C09126=1020.009,-60.580,383.207,-24.059,21.610,-43.700
C09127=1020.010,-60.243,383.182,-24.060,21.610,-43.695
C09128=1020.011,-59.906,383.156,-24.060,21.609,-43.691
C09129=1020.011,-59.569,383.131,-24.061,21.609,-43.686
C09130=1020.011,-59.234,383.106,-24.062,21.608,-43.680
C09131=1020.012,-58.898,383.081,-24.062,21.608,-43.676
C09132=1020.012,-58.562,383.056,-24.063,21.607,-43.671
C09133=1020.013,-58.228,383.030,-24.064,21.607,-43.666
C09134=1020.014,-57.893,383.005,-24.064,21.606,-43.662
C09135=1020.014,-57.559,382.981,-24.065,21.606,-43.656
C09136=1020.014,-57.225,382.955,-24.066,21.605,-43.652
C09137=1020.015,-56.892,382.930,-24.066,21.604,-43.647
C09138=1020.015,-56.558,382.905,-24.067,21.605,-43.642
C09139=1020.017,-56.225,382.880,-24.068,21.603,-43.637
C09140=1020.017,-55.892,382.855,-24.068,21.603,-43.632
C09141=1020.017,-55.559,382.830,-24.069,21.603,-43.627
C09142=1020.018,-55.226,382.805,-24.070,21.602,-43.623
C09143=1020.018,-54.894,382.780,-24.070,21.602,-43.618
C09144=1020.019,-54.562,382.755,-24.071,21.601,-43.613
C09145=1020.019,-54.229,382.729,-24.072,21.601,-43.608
C09146=1020.019,-53.896,382.704,-24.072,21.600,-43.603
C09147=1020.020,-53.565,382.679,-24.073,21.599,-43.599
C09148=1020.020,-53.232,382.654,-24.074,21.600,-43.594
C09149=1020.021,-52.900,382.629,-24.074,21.598,-43.589
C09150=1020.021,-52.568,382.604,-24.075,21.598,-43.584
C09151=1020.021,-52.235,382.579,-24.075,21.597,-43.579
C09152=1020.022,-51.903,382.554,-24.076,21.597,-43.575
C09153=1020.022,-51.571,382.528,-24.077,21.597,-43.570
C09154=1020.022,-51.238,382.503,-24.077,21.596,-43.566
C09155=1020.023,-50.906,382.478,-24.078,21.596,-43.560
C09156=1020.023,-50.524,382.449,-24.079,21.595,-43.555
C09157=1020.012,-29.274,380.804,-24.119,21.564,-43.254
C09158=1020.012,-28.955,380.779,-24.119,21.563,-43.250
C09159=1020.011,-28.621,380.753,-24.120,21.563,-43.245
C09160=1020.011,-28.288,380.727,-24.120,21.562,-43.241
C09161=1020.010,-27.956,380.700,-24.121,21.562,-43.236
C09162=1020.009,-27.623,380.673,-24.122,21.562,-43.232
C09163=1020.009,-27.291,380.647,-24.123,21.562,-43.227
C09164=1020.008,-26.957,380.622,-24.123,21.560,-43.223
C09165=1020.007,-26.625,380.595,-24.124,21.560,-43.217
C09166=1020.007,-26.292,380.569,-24.124,21.560,-43.214
C09167=1020.006,-25.960,380.542,-24.125,21.559,-43.208
C09168=1020.005,-25.627,380.516,-24.126,21.559,-43.204
C09169=1020.004,-25.294,380.490,-24.126,21.559,-43.199
C09170=1020.004,-24.960,380.463,-24.127,21.558,-43.195
C09171=1020.003,-24.628,380.437,-24.128,21.558,-43.190
C09172=1020.003,-24.295,380.410,-24.128,21.557,-43.186
C09173=1020.001,-23.963,380.384,-24.129,21.557,-43.181
C09174=1020.001,-23.630,380.357,-24.129,21.556,-43.177
C09175=1020.000,-23.297,380.332,-24.130,21.556,-43.171
C09176=1019.999,-22.964,380.305,-24.131,21.555,-43.168
C09177=1019.998,-22.632,380.279,-24.131,21.556,-43.162
C09178=1019.997,-22.299,380.252,-24.132,21.554,-43.158
C09179=1019.996,-21.966,380.225,-24.133,21.554,-43.153
C09180=1019.995,-21.633,380.198,-24.133,21.554,-43.149
C09181=1019.995,-21.301,380.172,-24.134,21.553,-43.144
C09182=1019.993,-20.967,380.146,-24.134,21.552,-43.140
C09183=1019.993,-20.634,380.119,-24.135,21.553,-43.135
C09184=1019.992,-20.301,380.093,-24.136,21.552,-43.131
C09185=1019.991,-19.969,380.066,-24.136,21.551,-43.127
C09186=1019.990,-19.636,380.039,-24.137,21.551,-43.122
C09187=1019.990,-19.464,380.025,-24.137,21.550,-43.118
C09188=1019.989,-19.048,379.992,-24.138,21.550,-43.112
C09189=1019.987,-18.800,379.973,-24.139,21.550,-43.109
C09190=1019.987,-18.538,379.952,-24.139,21.550,-43.107
C09191=1019.986,-18.276,379.931,-24.139,21.549,-43.105
C09192=1019.985,-18.029,379.911,-24.139,21.548,-43.103
C09193=1019.984,-17.807,379.893,-24.140,21.549,-43.100
C09194=1019.984,-17.442,379.864,-24.141,21.548,-43.092
C09195=1019.982,-17.109,379.837,-24.141,21.547,-43.088
C09196=1019.981,-16.776,379.811,-24.142,21.547,-43.083
C09197=1019.980,-16.442,379.783,-24.142,21.547,-43.079
C09198=1019.979,-16.109,379.757,-24.143,21.546,-43.074
C09199=1019.978,-15.775,379.730,-24.144,21.546,-43.070
C09200=1019.977,-15.439,379.703,-24.145,21.546,-43.065
C09201=1019.976,-15.103,379.676,-24.145,21.545,-43.061
C09202=1019.975,-14.765,379.649,-24.146,21.544,-43.055
C09203=1019.974,-14.425,379.622,-24.146,21.544,-43.052
C09204=1019.972,-14.083,379.593,-24.147,21.544,-43.046
C09205=1019.970,-13.739,379.566,-24.147,21.543,-43.042
C09206=1019.970,-13.392,379.538,-24.148,21.543,-43.037
C09207=1019.969,-13.044,379.510,-24.149,21.542,-43.033
C09208=1019.967,-12.694,379.481,-24.149,21.542,-43.028
C09209=1019.966,-12.342,379.453,-24.150,21.541,-43.024
C09210=1019.965,-11.989,379.425,-24.151,21.541,-43.019
C09211=1019.964,-11.633,379.396,-24.151,21.540,-43.014
C09212=1019.962,-11.277,379.367,-24.152,21.540,-43.009
C09213=1019.961,-10.919,379.338,-24.152,21.539,-43.006
C09214=1019.959,-10.560,379.309,-24.153,21.539,-43.000
C09215=1019.958,-10.200,379.280,-24.154,21.539,-42.995
C09216=1019.957,-9.839,379.251,-24.154,21.538,-42.991
C09217=1019.955,-9.478,379.222,-24.155,21.538,-42.985
C09218=1019.953,-9.115,379.192,-24.156,21.537,-42.982
C09219=1019.951,-8.753,379.163,-24.156,21.536,-42.976
C09220=1019.951,-8.390,379.134,-24.157,21.536,-42.971
C09221=1019.949,-8.027,379.104,-24.158,21.536,-42.967
C09222=1019.947,-7.664,379.074,-24.158,21.535,-42.961
C09223=1019.946,-7.298,379.045,-24.159,21.535,-42.956
C09224=1019.944,-6.929,379.014,-24.160,21.534,-42.952
C09225=1019.942,-6.557,378.984,-24.160,21.534,-42.947
C09226=1019.941,-6.183,378.954,-24.161,21.533,-42.941
C09227=1019.939,-5.806,378.923,-24.162,21.533,-42.937
C09228=1019.937,-5.431,378.893,-24.163,21.533,-42.932
C09229=1019.936,-5.058,378.862,-24.163,21.532,-42.928
C09230=1019.934,-4.687,378.831,-24.164,21.532,-42.923
C09231=1019.932,-4.322,378.802,-24.164,21.531,-42.919
C09232=1019.931,-3.961,378.772,-24.165,21.530,-42.913
C09233=1019.929,-3.602,378.743,-24.166,21.531,-42.908
C09234=1019.927,-3.249,378.714,-24.166,21.529,-42.904
C09235=1019.926,-2.896,378.685,-24.167,21.529,-42.899
C09236=1019.924,-2.544,378.656,-24.167,21.529,-42.895
C09237=1019.922,-2.195,378.627,-24.168,21.529,-42.890
C09238=1019.920,-1.846,378.599,-24.169,21.528,-42.886
C09239=1019.918,-1.500,378.571,-24.169,21.528,-42.880
C09240=1019.917,-1.155,378.542,-24.170,21.527,-42.877
C09241=1019.916,-0.811,378.514,-24.170,21.527,-42.873
C09242=1019.914,-0.469,378.486,-24.171,21.526,-42.867
C09243=1019.912,-0.129,378.458,-24.172,21.526,-42.864
C09244=1019.910,0.209,378.430,-24.172,21.526,-42.858
C09245=1019.909,0.546,378.403,-24.173,21.525,-42.855
C09246=1019.907,0.882,378.375,-24.173,21.525,-42.851
C09247=1019.906,1.217,378.348,-24.174,21.525,-42.846
C09248=1019.903,1.551,378.320,-24.175,21.524,-42.842
C09249=1019.901,1.885,378.293,-24.175,21.523,-42.838
C09250=1019.900,2.215,378.266,-24.176,21.523,-42.834
C09251=1019.898,2.528,378.239,-24.176,21.523,-42.831
C09252=1019.897,2.816,378.215,-24.177,21.522,-42.827
C09253=1019.895,3.085,378.194,-24.177,21.522,-42.823
C09254=1019.894,3.347,378.172,-24.178,21.522,-42.818
C09255=1019.892,3.616,378.150,-24.179,21.521,-42.814
C09256=1019.890,3.905,378.126,-24.179,21.521,-42.810
C09257=1019.889,4.218,378.100,-24.179,21.520,-42.807
C09258=1019.887,4.548,378.073,-24.180,21.521,-42.803
C09259=1019.884,4.880,378.045,-24.180,21.519,-42.799
C09260=1019.883,5.211,378.018,-24.181,21.519,-42.795
C09261=1019.881,5.541,377.990,-24.181,21.518,-42.792
C09262=1019.879,5.872,377.963,-24.182,21.519,-42.786
C09263=1019.877,6.202,377.936,-24.183,21.518,-42.783
C09264=1019.876,6.531,377.909,-24.183,21.518,-42.779
C09265=1019.873,6.860,377.881,-24.184,21.518,-42.774
C09266=1019.872,7.189,377.854,-24.185,21.517,-42.770
C09267=1019.870,7.516,377.827,-24.185,21.517,-42.766
C09268=1019.867,7.842,377.799,-24.186,21.516,-42.762
C09269=1019.866,8.165,377.773,-24.186,21.516,-42.759
C09270=1019.864,8.486,377.746,-24.186,21.515,-42.755
C09271=1019.862,8.804,377.720,-24.187,21.516,-42.750
C09272=1019.860,9.120,377.694,-24.188,21.515,-42.746
C09273=1019.858,9.436,377.668,-24.188,21.515,-42.742
C09274=1019.856,9.750,377.641,-24.189,21.514,-42.738
C09275=1019.854,10.065,377.615,-24.190,21.514,-42.733
C09276=1019.852,10.380,377.589,-24.190,21.514,-42.730
C09277=1019.850,10.698,377.562,-24.191,21.513,-42.726
C09278=1019.848,11.016,377.535,-24.191,21.513,-42.722
C09279=1019.846,11.337,377.509,-24.192,21.512,-42.718
C09280=1019.843,11.659,377.482,-24.192,21.512,-42.715
C09281=1019.842,11.982,377.455,-24.193,21.511,-42.711
C09282=1019.840,12.306,377.428,-24.193,21.511,-42.707
C09283=1019.837,12.630,377.401,-24.194,21.511,-42.702
C09284=1019.835,12.953,377.374,-24.194,21.510,-42.698
C09285=1019.833,13.277,377.346,-24.195,21.510,-42.694
C09286=1019.831,13.601,377.320,-24.195,21.509,-42.691
C09287=1019.828,13.924,377.292,-24.196,21.509,-42.687
C09288=1019.827,14.249,377.265,-24.197,21.509,-42.682
C09289=1019.825,14.574,377.238,-24.197,21.509,-42.678
C09290=1019.823,14.899,377.211,-24.198,21.508,-42.674
C09291=1019.820,15.224,377.184,-24.198,21.508,-42.670
C09292=1019.818,15.550,377.156,-24.199,21.507,-42.667
C09293=1019.816,15.877,377.129,-24.199,21.507,-42.663
C09294=1019.813,16.204,377.102,-24.200,21.507,-42.658
C09295=1019.811,16.531,377.074,-24.200,21.506,-42.654
C09296=1019.809,16.859,377.047,-24.201,21.506,-42.650
C09297=1019.807,17.188,377.019,-24.201,21.505,-42.646
C09298=1019.804,17.517,376.992,-24.202,21.505,-42.643
C09299=1019.801,17.847,376.964,-24.202,21.504,-42.639
C09300=1019.799,18.177,376.936,-24.203,21.504,-42.634
C09301=1019.797,18.508,376.908,-24.204,21.504,-42.630
C09302=1019.794,18.839,376.880,-24.204,21.503,-42.626
C09303=1019.792,19.171,376.853,-24.205,21.503,-42.622
C09304=1019.790,19.504,376.824,-24.205,21.502,-42.619
C09305=1019.787,19.851,376.795,-24.206,21.503,-42.613
C09306=1019.784,20.269,376.760,-24.207,21.502,-42.608
C09307=1019.782,20.505,376.739,-24.207,21.502,-42.604
C09308=1019.781,20.752,376.719,-24.207,21.502,-42.603
C09309=1019.779,21.000,376.698,-24.208,21.502,-42.601
C09310=1019.776,21.241,376.678,-24.208,21.502,-42.599
C09311=1019.775,21.469,376.658,-24.208,21.501,-42.597
C09312=1019.773,21.676,376.641,-24.209,21.501,-42.593
C09313=1019.771,22.033,376.611,-24.209,21.500,-42.588
C09314=1019.768,22.357,376.583,-24.210,21.501,-42.584
C09315=1019.766,22.651,376.558,-24.210,21.500,-42.582
C09316=1019.764,22.904,376.537,-24.210,21.499,-42.580
C09317=1019.761,23.313,376.502,-24.211,21.499,-42.573
C09318=1019.758,23.722,376.468,-24.212,21.498,-42.565
C09319=1019.756,23.974,376.446,-24.213,21.498,-42.562
C09320=1019.753,24.268,376.422,-24.213,21.498,-42.560
C09321=1019.750,24.595,376.394,-24.213,21.497,-42.558
C09322=1019.748,24.929,376.366,-24.214,21.497,-42.553
C09323=1019.746,25.263,376.337,-24.215,21.497,-42.549
C09324=1019.743,25.598,376.309,-24.215,21.496,-42.545
C09325=1019.740,25.931,376.281,-24.216,21.496,-42.541
C09326=1019.737,26.266,376.252,-24.216,21.495,-42.538
C09327=1019.735,26.601,376.224,-24.217,21.495,-42.534
C09328=1019.732,26.935,376.195,-24.217,21.494,-42.530
C09329=1019.729,27.269,376.167,-24.218,21.494,-42.525
C09330=1019.726,27.604,376.139,-24.219,21.495,-42.522
C09331=1019.724,27.938,376.110,-24.219,21.494,-42.518
C09332=1019.721,28.273,376.081,-24.220,21.494,-42.514
C09333=1019.719,28.607,376.054,-24.220,21.493,-42.510
C09334=1019.715,28.941,376.025,-24.221,21.493,-42.507
C09335=1019.712,29.276,375.996,-24.221,21.492,-42.503
C09336=1019.710,29.610,375.968,-24.222,21.493,-42.498
C09337=1019.707,29.945,375.939,-24.222,21.492,-42.494
C09338=1019.704,30.279,375.910,-24.223,21.492,-42.490
C09339=1019.701,30.613,375.883,-24.223,21.491,-42.486
C09340=1019.698,30.948,375.854,-24.224,21.491,-42.483
C09341=1019.695,31.282,375.825,-24.224,21.490,-42.479
C09342=1019.692,31.618,375.796,-24.225,21.490,-42.475
C09343=1019.689,31.952,375.767,-24.225,21.489,-42.471
C09344=1019.687,32.287,375.740,-24.226,21.489,-42.468
C09345=1019.683,32.621,375.711,-24.226,21.489,-42.464
C09346=1019.681,32.955,375.682,-24.227,21.489,-42.459
C09347=1019.677,33.290,375.654,-24.228,21.489,-42.455
C09348=1019.674,33.625,375.625,-24.228,21.488,-42.452
C09349=1019.671,33.960,375.596,-24.229,21.488,-42.448
C09350=1019.668,34.294,375.567,-24.229,21.487,-42.444
C09351=1019.666,34.629,375.538,-24.230,21.487,-42.440
C09352=1019.662,34.964,375.510,-24.230,21.486,-42.437
C09353=1019.660,35.298,375.481,-24.231,21.486,-42.433
C09354=1019.656,35.633,375.453,-24.231,21.485,-42.429
C09355=1019.653,35.967,375.424,-24.232,21.486,-42.426
C09356=1019.650,36.302,375.395,-24.232,21.485,-42.422
C09357=1019.647,36.637,375.367,-24.233,21.485,-42.418
C09358=1019.644,36.971,375.338,-24.234,21.485,-42.413
C09359=1019.641,37.307,375.309,-24.234,21.485,-42.409
C09360=1019.638,37.641,375.280,-24.235,21.484,-42.405
C09361=1019.635,37.976,375.252,-24.235,21.484,-42.402
C09362=1019.632,38.311,375.223,-24.236,21.483,-42.398
C09363=1019.628,38.645,375.193,-24.236,21.483,-42.395
C09364=1019.625,38.981,375.165,-24.237,21.483,-42.391
C09365=1019.622,39.315,375.136,-24.237,21.483,-42.387
C09366=1019.618,39.649,375.108,-24.238,21.482,-42.383
C09367=1019.615,39.984,375.078,-24.238,21.482,-42.380
C09368=1019.612,40.319,375.050,-24.239,21.481,-42.376
C09369=1019.609,40.654,375.021,-24.239,21.481,-42.372
C09370=1019.606,40.989,374.993,-24.240,21.481,-42.369
C09371=1019.602,41.324,374.963,-24.240,21.481,-42.365
C09372=1019.599,41.658,374.934,-24.241,21.480,-42.361
C09373=1019.596,41.993,374.906,-24.241,21.480,-42.357
C09374=1019.592,42.328,374.876,-24.242,21.479,-42.354
C09375=1019.589,42.663,374.848,-24.242,21.479,-42.350
C09376=1019.586,42.998,374.818,-24.243,21.479,-42.347
C09377=1019.582,43.333,374.790,-24.243,21.479,-42.343
C09378=1019.579,43.668,374.760,-24.244,21.478,-42.339
C09379=1019.576,44.003,374.732,-24.244,21.478,-42.335
C09380=1019.572,44.338,374.702,-24.245,21.477,-42.332
C09381=1019.569,44.673,374.674,-24.245,21.477,-42.328
C09382=1019.565,45.008,374.644,-24.246,21.477,-42.325
C09383=1019.562,45.343,374.616,-24.246,21.477,-42.321
C09384=1019.558,45.678,374.586,-24.247,21.476,-42.317
C09385=1019.556,46.012,374.557,-24.247,21.476,-42.313
C09386=1019.552,46.348,374.528,-24.248,21.475,-42.309
C09387=1019.547,46.682,374.499,-24.248,21.475,-42.306
C09388=1019.544,47.017,374.471,-24.249,21.475,-42.302
C09389=1019.541,47.352,374.441,-24.249,21.475,-42.299
C09390=1019.538,47.687,374.413,-24.250,21.474,-42.295
C09391=1019.534,48.022,374.383,-24.250,21.474,-42.291
C09392=1019.530,48.357,374.354,-24.251,21.473,-42.287
C09393=1019.526,48.692,374.325,-24.251,21.473,-42.284
C09394=1019.523,49.027,374.297,-24.252,21.473,-42.280
C09395=1019.520,49.362,374.267,-24.252,21.473,-42.277
C09396=1019.516,49.697,374.238,-24.253,21.472,-42.273
C09397=1019.512,50.032,374.208,-24.253,21.472,-42.269
C09398=1019.509,50.367,374.180,-24.254,21.472,-42.266
C09399=1019.505,50.702,374.150,-24.254,21.471,-42.262
C09400=1019.502,51.037,374.121,-24.255,21.471,-42.258
C09401=1019.498,51.372,374.092,-24.255,21.471,-42.254
C09402=1019.494,51.707,374.062,-24.256,21.471,-42.251
C09403=1019.490,52.042,374.033,-24.256,21.470,-42.247
C09404=1019.487,52.377,374.004,-24.257,21.470,-42.244
C09405=1019.483,52.712,373.976,-24.257,21.470,-42.240
C09406=1019.479,53.046,373.946,-24.258,21.469,-42.238
C09407=1019.475,53.382,373.917,-24.258,21.469,-42.234
C09408=1019.472,53.717,373.888,-24.259,21.468,-42.230
C09409=1019.468,54.052,373.859,-24.259,21.468,-42.227
C09410=1019.464,54.387,373.829,-24.260,21.468,-42.223
C09411=1019.460,54.722,373.800,-24.260,21.468,-42.220
C09412=1019.457,55.057,373.771,-24.261,21.467,-42.216
C09413=1019.453,55.392,373.741,-24.261,21.467,-42.212
C09414=1019.449,55.727,373.712,-24.262,21.467,-42.209
C09415=1019.446,56.062,373.682,-24.262,21.467,-42.205
C09416=1019.441,56.397,373.654,-24.263,21.466,-42.201
C09417=1019.437,56.732,373.624,-24.263,21.466,-42.197
C09418=1019.433,57.067,373.595,-24.264,21.466,-42.194
C09419=1019.429,57.402,373.565,-24.264,21.465,-42.192
C09420=1019.425,57.738,373.536,-24.264,21.465,-42.188
C09421=1019.422,58.073,373.507,-24.265,21.464,-42.184
C09422=1019.418,58.407,373.477,-24.266,21.465,-42.181
C09423=1019.414,58.742,373.448,-24.266,21.464,-42.177
C09424=1019.409,59.077,373.418,-24.267,21.464,-42.173
C09425=1019.405,59.413,373.389,-24.267,21.464,-42.170
C09426=1019.402,59.747,373.360,-24.268,21.464,-42.166
C09427=1019.398,60.083,373.331,-24.268,21.463,-42.163
C09428=1019.393,60.418,373.300,-24.268,21.462,-42.160
C09429=1019.389,60.752,373.271,-24.269,21.462,-42.157
C09430=1019.385,61.087,373.242,-24.269,21.462,-42.153
C09431=1019.382,61.422,373.213,-24.270,21.461,-42.149
C09432=1019.377,61.758,373.183,-24.270,21.462,-42.146
C09433=1019.373,62.093,373.154,-24.271,21.461,-42.142
C09434=1019.369,62.427,373.124,-24.271,21.461,-42.139
C09435=1019.365,62.764,373.095,-24.272,21.460,-42.135
C09436=1019.360,63.160,373.060,-24.272,21.460,-42.131
C09437=1019.357,63.384,373.040,-24.273,21.461,-42.130
C09438=1019.357,63.602,373.019,-24.273,21.460,-42.128
C09439=1019.356,63.976,372.984,-24.274,21.460,-42.124
C09440=1019.355,64.332,372.951,-24.274,21.459,-42.120
C09441=1019.354,64.718,372.914,-24.274,21.459,-42.116
C09442=1019.353,65.113,372.877,-24.275,21.458,-42.113
C09443=1019.352,65.491,372.842,-24.276,21.459,-42.108
C09444=1019.351,65.845,372.808,-24.276,21.457,-42.105
C09445=1019.350,66.184,372.776,-24.277,21.458,-42.102
C09446=1019.349,66.517,372.745,-24.277,21.457,-42.098
C09447=1019.348,66.852,372.713,-24.278,21.457,-42.094
C09448=1019.347,67.189,372.681,-24.278,21.457,-42.091
C09449=1019.346,67.527,372.650,-24.279,21.457,-42.087
C09450=1019.345,67.865,372.618,-24.279,21.456,-42.085
C09451=1019.344,68.205,372.586,-24.279,21.456,-42.082
C09452=1019.343,68.545,372.553,-24.280,21.456,-42.078
C09453=1019.342,68.886,372.521,-24.280,21.455,-42.074
C09454=1019.342,69.228,372.488,-24.281,21.456,-42.071
C09455=1019.340,69.572,372.456,-24.281,21.455,-42.067
C09456=1019.340,69.915,372.424,-24.282,21.455,-42.063
C09457=1019.338,70.259,372.391,-24.282,21.454,-42.061
C09458=1019.337,70.604,372.358,-24.283,21.454,-42.058
C09459=1019.337,70.949,372.325,-24.283,21.453,-42.054
C09460=1019.335,71.293,372.293,-24.284,21.454,-42.051
C09461=1019.335,71.638,372.260,-24.284,21.453,-42.047
C09462=1019.333,71.982,372.227,-24.285,21.453,-42.043
C09463=1019.333,72.328,372.195,-24.285,21.453,-42.041
C09464=1019.332,72.674,372.162,-24.285,21.452,-42.037
C09465=1019.330,73.022,372.128,-24.286,21.452,-42.034
C09466=1019.329,73.372,372.095,-24.286,21.451,-42.030
C09467=1019.328,73.723,372.062,-24.287,21.452,-42.027
C09468=1019.326,74.077,372.028,-24.288,21.451,-42.023
C09469=1019.326,74.432,371.994,-24.288,21.451,-42.019
C09470=1019.325,74.788,371.960,-24.288,21.451,-42.017
C09471=1019.325,75.147,371.926,-24.289,21.450,-42.013
C09472=1019.323,75.504,371.892,-24.289,21.450,-42.010
C09473=1019.322,75.858,371.858,-24.290,21.450,-42.006
C09474=1019.320,76.207,371.825,-24.290,21.449,-42.004
C09475=1019.320,76.548,371.792,-24.291,21.449,-42.001
C09476=1019.319,76.884,371.760,-24.291,21.449,-41.997
C09477=1019.318,77.215,371.728,-24.292,21.449,-41.994
C09478=1019.317,77.542,371.697,-24.292,21.449,-41.990
C09479=1019.316,77.865,371.666,-24.292,21.448,-41.987
C09480=1019.315,78.188,371.634,-24.293,21.448,-41.984
C09481=1019.314,78.513,371.604,-24.293,21.448,-41.980
C09482=1019.313,78.841,371.573,-24.294,21.447,-41.977
C09483=1019.312,79.174,371.541,-24.295,21.448,-41.973
C09484=1019.311,79.512,371.509,-24.295,21.446,-41.971
C09485=1019.309,79.858,371.475,-24.295,21.447,-41.968
C09486=1019.309,80.208,371.441,-24.296,21.446,-41.964
C09487=1019.307,80.563,371.407,-24.296,21.446,-41.962
C09488=1019.306,80.921,371.373,-24.297,21.446,-41.958
C09489=1019.306,81.277,371.339,-24.297,21.445,-41.955
C09490=1019.304,81.633,371.305,-24.298,21.446,-41.951
C09491=1019.303,81.988,371.270,-24.298,21.445,-41.947
C09492=1019.302,82.343,371.236,-24.298,21.444,-41.945
C09493=1019.301,82.697,371.202,-24.299,21.444,-41.942
C09494=1019.299,83.050,371.168,-24.299,21.444,-41.938
C09495=1019.298,83.401,371.134,-24.300,21.444,-41.935
C09496=1019.297,83.752,371.100,-24.300,21.444,-41.931
C09497=1019.296,84.102,371.066,-24.301,21.443,-41.929
C09498=1019.295,84.451,371.033,-24.301,21.443,-41.925
C09499=1019.293,84.799,370.999,-24.302,21.443,-41.922
C09500=1019.293,85.146,370.966,-24.302,21.443,-41.918
C09501=1019.291,85.491,370.932,-24.302,21.442,-41.916
C09502=1019.290,85.836,370.899,-24.303,21.442,-41.912
C09503=1019.289,86.178,370.866,-24.303,21.442,-41.909
C09504=1019.288,86.520,370.833,-24.304,21.441,-41.906
C09505=1019.287,86.861,370.800,-24.304,21.441,-41.903
C09506=1019.286,87.200,370.767,-24.305,21.441,-41.899
C09507=1019.285,87.537,370.735,-24.305,21.441,-41.898
C09508=1019.284,87.869,370.702,-24.305,21.440,-41.894
C09509=1019.283,88.196,370.671,-24.306,21.441,-41.890
C09510=1019.282,88.519,370.639,-24.306,21.439,-41.888
C09511=1019.280,88.839,370.608,-24.307,21.440,-41.885
C09512=1019.280,89.160,370.577,-24.307,21.439,-41.881
C09513=1019.279,89.485,370.545,-24.308,21.439,-41.879
C09514=1019.278,89.814,370.513,-24.308,21.440,-41.876
C09515=1019.277,90.148,370.481,-24.308,21.438,-41.874
C09516=1019.275,90.482,370.449,-24.309,21.439,-41.870
C09517=1019.274,90.816,370.416,-24.309,21.438,-41.866
C09518=1019.273,91.150,370.383,-24.310,21.438,-41.865
C09519=1019.273,91.485,370.351,-24.310,21.438,-41.861
C09520=1019.271,91.819,370.318,-24.311,21.438,-41.857
C09521=1019.270,92.153,370.286,-24.311,21.437,-41.855
C09522=1019.269,92.489,370.253,-24.311,21.437,-41.852
C09523=1019.267,92.823,370.221,-24.312,21.436,-41.849
C09524=1019.266,93.157,370.189,-24.312,21.437,-41.846
C09525=1019.265,93.491,370.156,-24.313,21.436,-41.842
C09526=1019.264,93.826,370.123,-24.313,21.436,-41.841
C09527=1019.263,94.160,370.090,-24.314,21.436,-41.837
C09528=1019.261,94.494,370.058,-24.314,21.436,-41.833
C09529=1019.260,94.829,370.025,-24.314,21.436,-41.832
C09530=1019.260,95.163,369.992,-24.315,21.435,-41.828
C09531=1019.259,95.497,369.960,-24.315,21.435,-41.826
C09532=1019.257,95.832,369.927,-24.316,21.435,-41.822
C09533=1019.256,96.166,369.895,-24.316,21.435,-41.819
C09534=1019.255,96.500,369.861,-24.316,21.434,-41.817
C09535=1019.254,96.835,369.828,-24.317,21.434,-41.813
C09536=1019.252,97.169,369.796,-24.317,21.434,-41.811
C09537=1019.252,97.502,369.763,-24.318,21.434,-41.808
C09538=1019.250,97.837,369.731,-24.318,21.433,-41.806
C09539=1019.250,98.171,369.697,-24.318,21.433,-41.802
C09540=1019.248,98.506,369.665,-24.319,21.433,-41.799
C09541=1019.247,98.840,369.632,-24.319,21.432,-41.796
C09542=1019.245,99.174,369.599,-24.320,21.433,-41.793
C09543=1019.244,99.508,369.566,-24.320,21.432,-41.791
C09544=1019.243,99.842,369.533,-24.320,21.432,-41.787
C09545=1019.242,100.177,369.500,-24.321,21.432,-41.785
C09546=1019.241,100.510,369.468,-24.321,21.431,-41.782
C09547=1019.240,100.844,369.435,-24.322,21.432,-41.778
C09548=1019.239,101.178,369.402,-24.322,21.431,-41.776
C09549=1019.237,101.513,369.370,-24.323,21.431,-41.773
C09550=1019.237,101.847,369.336,-24.323,21.431,-41.771
C09551=1019.235,102.181,369.303,-24.323,21.430,-41.767
C09552=1019.234,102.515,369.270,-24.324,21.430,-41.765
C09553=1019.233,102.849,369.238,-24.324,21.431,-41.762
C09554=1019.231,103.183,369.205,-24.324,21.429,-41.760
C09555=1019.230,103.517,369.172,-24.325,21.430,-41.756
C09556=1019.229,103.852,369.138,-24.325,21.429,-41.752
C09557=1019.228,104.186,369.105,-24.326,21.429,-41.751
C09558=1019.227,104.520,369.073,-24.326,21.430,-41.747
C09559=1019.225,104.854,369.039,-24.326,21.428,-41.745
C09560=1019.224,105.188,369.007,-24.327,21.429,-41.742
C09561=1019.223,105.522,368.974,-24.327,21.428,-41.739
C09562=1019.222,105.855,368.941,-24.328,21.428,-41.736
C09563=1019.221,106.191,368.908,-24.328,21.428,-41.734
C09564=1019.220,106.524,368.874,-24.328,21.427,-41.730
C09565=1019.218,106.858,368.841,-24.329,21.427,-41.728
C09566=1019.217,107.192,368.809,-24.329,21.428,-41.725
C09567=1019.216,107.526,368.775,-24.329,21.427,-41.723
C09568=1019.215,107.860,368.742,-24.330,21.427,-41.719
C09569=1019.213,108.193,368.709,-24.330,21.427,-41.718
C09570=1019.212,108.529,368.676,-24.331,21.426,-41.714
C09571=1019.211,108.862,368.643,-24.331,21.426,-41.712
C09572=1019.210,109.196,368.610,-24.332,21.426,-41.708
C09573=1019.208,109.530,368.576,-24.332,21.425,-41.706
C09574=1019.207,109.864,368.543,-24.332,21.426,-41.703
C09575=1019.206,110.198,368.510,-24.333,21.425,-41.701
C09576=1019.205,110.532,368.477,-24.333,21.425,-41.697
C09577=1019.204,110.866,368.443,-24.333,21.425,-41.695
C09578=1019.203,111.200,368.410,-24.334,21.424,-41.692
C09579=1019.201,111.534,368.377,-24.334,21.424,-41.690
C09580=1019.200,111.868,368.344,-24.335,21.425,-41.686
C09581=1019.199,112.202,368.311,-24.335,21.423,-41.684
C09582=1019.197,112.536,368.277,-24.335,21.424,-41.681
C09583=1019.196,112.870,368.244,-24.336,21.424,-41.679
C09584=1019.195,113.204,368.211,-24.336,21.423,-41.675
C09585=1019.194,113.538,368.177,-24.336,21.423,-41.673
C09586=1019.193,113.871,368.144,-24.337,21.423,-41.670
C09587=1019.192,114.205,368.111,-24.337,21.422,-41.668
C09588=1019.190,114.539,368.077,-24.338,21.423,-41.664
C09589=1019.189,114.873,368.044,-24.338,21.422,-41.662
C09590=1019.188,115.208,368.011,-24.338,21.421,-41.660
C09591=1019.186,115.542,367.978,-24.339,21.422,-41.657
C09592=1019.184,115.876,367.944,-24.339,21.422,-41.655
C09593=1019.183,116.209,367.911,-24.340,21.422,-41.652
C09594=1019.183,116.544,367.877,-24.340,21.421,-41.649
C09595=1019.182,116.877,367.844,-24.340,21.421,-41.646
C09596=1019.180,117.211,367.811,-24.341,21.421,-41.644
C09597=1019.178,117.545,367.777,-24.341,21.421,-41.640
C09598=1019.177,117.879,367.744,-24.341,21.420,-41.638
C09599=1019.177,118.213,367.710,-24.342,21.421,-41.635
C09600=1019.175,118.547,367.676,-24.342,21.420,-41.633
C09601=1019.174,118.881,367.643,-24.342,21.419,-41.631
C09602=1019.172,119.215,367.610,-24.343,21.420,-41.628
C09603=1019.172,119.549,367.576,-24.343,21.419,-41.625
C09604=1019.170,119.883,367.542,-24.344,21.419,-41.622
C09605=1019.169,120.216,367.509,-24.344,21.419,-41.620
C09606=1019.168,120.550,367.475,-24.345,21.419,-41.617
C09607=1019.167,120.885,367.441,-24.345,21.418,-41.614
C09608=1019.165,121.219,367.408,-24.345,21.418,-41.613
C09609=1019.164,121.552,367.375,-24.346,21.418,-41.609
C09610=1019.162,121.886,367.341,-24.346,21.417,-41.607
C09611=1019.162,122.221,367.307,-24.346,21.418,-41.604
C09612=1019.160,122.555,367.274,-24.347,21.418,-41.602
C09613=1019.159,122.889,367.240,-24.347,21.418,-41.598
C09614=1019.158,123.222,367.206,-24.347,21.417,-41.596
C09615=1019.156,123.556,367.172,-24.348,21.417,-41.594
C09616=1019.155,123.890,367.139,-24.348,21.417,-41.591
C09617=1019.153,124.224,367.105,-24.348,21.417,-41.589
C09618=1019.153,124.559,367.072,-24.349,21.416,-41.585
C09619=1019.152,124.892,367.038,-24.349,21.416,-41.583
C09620=1019.150,125.226,367.005,-24.349,21.416,-41.581
C09621=1019.149,125.560,366.970,-24.350,21.416,-41.578
C09622=1019.147,125.894,366.936,-24.350,21.415,-41.576
C09623=1019.146,126.228,366.903,-24.351,21.416,-41.572
C09624=1019.145,126.563,366.869,-24.351,21.415,-41.571
C09625=1019.144,126.896,366.836,-24.351,21.415,-41.569
C09626=1019.142,127.230,366.801,-24.352,21.415,-41.565
C09627=1019.142,127.564,366.768,-24.352,21.415,-41.563
C09628=1019.140,127.898,366.734,-24.352,21.414,-41.561
C09629=1019.139,128.233,366.700,-24.353,21.415,-41.558
C09630=1019.137,128.567,366.666,-24.353,21.414,-41.555
C09631=1019.136,128.900,366.633,-24.354,21.414,-41.552
C09632=1019.135,129.234,366.598,-24.354,21.414,-41.550
C09633=1019.134,129.568,366.565,-24.354,21.414,-41.548
C09634=1019.132,129.903,366.531,-24.355,21.413,-41.545
C09635=1019.131,130.236,366.496,-24.355,21.413,-41.543
C09636=1019.130,130.571,366.463,-24.355,21.413,-41.541
C09637=1019.128,130.905,366.429,-24.356,21.413,-41.538
C09638=1019.128,131.239,366.395,-24.356,21.412,-41.535
C09639=1019.126,131.573,366.361,-24.356,21.412,-41.532
C09640=1019.124,131.907,366.327,-24.357,21.412,-41.530
C09641=1019.124,132.241,366.293,-24.357,21.412,-41.528
C09642=1019.122,132.575,366.259,-24.357,21.412,-41.525
C09643=1019.121,132.909,366.225,-24.358,21.411,-41.523
C09644=1019.120,133.244,366.191,-24.358,21.411,-41.521
C09645=1019.119,133.577,366.157,-24.358,21.411,-41.517
C09646=1019.117,133.912,366.122,-24.359,21.411,-41.515
C09647=1019.116,134.246,366.089,-24.359,21.410,-41.513
C09648=1019.115,134.580,366.054,-24.359,21.411,-41.510
C09649=1019.113,134.914,366.021,-24.360,21.410,-41.508
C09650=1019.113,135.248,365.987,-24.360,21.410,-41.506
C09651=1019.111,135.582,365.952,-24.361,21.411,-41.503
C09652=1019.110,135.904,365.920,-24.361,21.410,-41.501
C09653=1019.109,136.204,365.889,-24.361,21.410,-41.499
C09654=1019.108,136.484,365.860,-24.361,21.410,-41.497
C09655=1019.106,136.749,365.833,-24.361,21.409,-41.495
C09656=1019.106,137.014,365.806,-24.362,21.409,-41.491
C09657=1019.105,137.290,365.778,-24.362,21.409,-41.490
C09658=1019.103,137.587,365.747,-24.363,21.409,-41.488
C09659=1019.102,137.909,365.714,-24.363,21.408,-41.486
C09660=1019.101,138.250,365.680,-24.363,21.408,-41.484
C09661=1019.100,138.606,365.643,-24.364,21.408,-41.480
C09662=1019.098,139.018,365.601,-24.364,21.408,-41.477
C09663=1019.097,139.245,365.578,-24.364,21.408,-41.475
C09664=1019.096,139.483,365.553,-24.365,21.408,-41.473
C09665=1019.095,139.725,365.528,-24.365,21.408,-41.473
C09666=1019.095,139.966,365.504,-24.365,21.408,-41.471
C09667=1019.094,140.198,365.480,-24.365,21.408,-41.470
C09668=1019.093,140.419,365.458,-24.365,21.407,-41.469
C09669=1019.091,140.812,365.417,-24.366,21.407,-41.465
C09670=1019.090,141.157,365.382,-24.366,21.407,-41.462
C09671=1019.089,141.496,365.347,-24.367,21.407,-41.460
C09672=1019.088,141.835,365.312,-24.367,21.407,-41.457
C09673=1019.086,142.175,365.277,-24.367,21.406,-41.455
C09674=1019.085,142.516,365.242,-24.368,21.406,-41.453
C09675=1019.084,142.858,365.207,-24.368,21.407,-41.449
C09676=1019.083,143.200,365.172,-24.368,21.406,-41.448
C09677=1019.081,143.543,365.136,-24.369,21.405,-41.445
C09678=1019.080,143.885,365.101,-24.369,21.406,-41.442
C09679=1019.079,144.230,365.066,-24.369,21.405,-41.440
C09680=1019.078,144.573,365.031,-24.370,21.405,-41.438
C09681=1019.076,144.917,364.995,-24.370,21.406,-41.435
C09682=1019.075,145.262,364.959,-24.370,21.405,-41.432
C09683=1019.074,145.608,364.924,-24.371,21.404,-41.431
C09684=1019.072,145.954,364.888,-24.371,21.405,-41.427
C09685=1019.071,146.300,364.853,-24.371,21.405,-41.425
C09686=1019.069,146.646,364.816,-24.372,21.404,-41.424
C09687=1019.059,146.992,364.786,-24.372,21.404,-41.420
C09688=1019.038,147.337,364.763,-24.372,21.404,-41.418
C09689=1019.413,147.364,364.529,-24.372,21.404,-41.418
C09690=1019.435,147.019,364.552,-24.372,21.404,-41.420
C09691=1019.446,146.673,364.581,-24.372,21.404,-41.424
C09692=1019.448,146.327,364.617,-24.371,21.405,-41.425
C09693=1019.450,145.981,364.652,-24.371,21.405,-41.427
C09694=1019.451,145.636,364.689,-24.371,21.404,-41.431
C09695=1019.452,145.290,364.724,-24.370,21.405,-41.432
C09696=1019.453,144.945,364.760,-24.370,21.406,-41.435
C09697=1019.455,144.600,364.795,-24.370,21.405,-41.438
C09698=1019.457,144.256,364.830,-24.369,21.405,-41.440
C09699=1019.457,143.913,364.866,-24.369,21.406,-41.442
C09700=1019.460,143.570,364.901,-24.369,21.405,-41.445
C09701=1019.461,143.227,364.936,-24.368,21.406,-41.448
C09702=1019.461,142.885,364.971,-24.368,21.407,-41.449
C09703=1019.463,142.544,365.007,-24.368,21.406,-41.453
C09704=1019.463,142.203,365.042,-24.367,21.406,-41.455
C09705=1019.465,141.863,365.077,-24.367,21.407,-41.457
C09706=1019.466,141.523,365.111,-24.367,21.407,-41.460
C09707=1019.468,141.184,365.146,-24.366,21.407,-41.462
C09708=1019.469,140.839,365.182,-24.366,21.407,-41.465
C09709=1019.470,140.446,365.222,-24.365,21.407,-41.469
C09710=1019.471,140.226,365.245,-24.365,21.408,-41.470
C09711=1019.472,139.993,365.269,-24.365,21.408,-41.471
C09712=1019.473,139.752,365.293,-24.365,21.408,-41.473
C09713=1019.474,139.510,365.319,-24.365,21.408,-41.473
C09714=1019.475,139.272,365.343,-24.364,21.408,-41.475
C09715=1019.475,139.044,365.366,-24.364,21.408,-41.477
C09716=1019.477,138.633,365.408,-24.364,21.408,-41.480
C09717=1019.479,138.277,365.445,-24.363,21.408,-41.484
C09718=1019.480,137.936,365.480,-24.363,21.408,-41.486
C09719=1019.481,137.614,365.512,-24.363,21.409,-41.488
C09720=1019.482,137.317,365.543,-24.362,21.409,-41.490
C09721=1019.483,137.040,365.571,-24.362,21.409,-41.491
C09722=1019.484,136.777,365.599,-24.361,21.409,-41.495
C09723=1019.485,136.511,365.625,-24.361,21.410,-41.497
C09724=1019.486,136.232,365.654,-24.361,21.410,-41.499
C09725=1019.487,135.932,365.684,-24.361,21.410,-41.501
C09726=1019.488,135.609,365.717,-24.361,21.411,-41.503
C09727=1019.490,135.276,365.752,-24.360,21.410,-41.506
C09728=1019.491,134.941,365.786,-24.360,21.410,-41.508
C09729=1019.492,134.607,365.819,-24.359,21.411,-41.510
C09730=1019.493,134.273,365.854,-24.359,21.410,-41.513
C09731=1019.495,133.939,365.888,-24.359,21.411,-41.515
C09732=1019.496,133.605,365.921,-24.358,21.411,-41.517
C09733=1019.497,133.270,365.955,-24.358,21.411,-41.521
C09734=1019.499,132.937,365.990,-24.358,21.411,-41.523
C09735=1019.499,132.602,366.024,-24.357,21.412,-41.525
C09736=1019.501,132.268,366.057,-24.357,21.412,-41.528
C09737=1019.502,131.934,366.092,-24.357,21.412,-41.530
C09738=1019.503,131.600,366.126,-24.356,21.412,-41.532
C09739=1019.505,131.266,366.160,-24.356,21.412,-41.535
C09740=1019.506,130.932,366.194,-24.356,21.413,-41.538
C09741=1019.507,130.598,366.228,-24.355,21.413,-41.541
C09742=1019.509,130.264,366.262,-24.355,21.413,-41.543
C09743=1019.509,129.929,366.295,-24.355,21.413,-41.545
C09744=1019.511,129.596,366.330,-24.354,21.414,-41.548
C09745=1019.512,129.261,366.363,-24.354,21.414,-41.550
C09746=1019.513,128.927,366.397,-24.354,21.414,-41.552
C09747=1019.515,128.594,366.430,-24.353,21.414,-41.555
C09748=1019.516,128.260,366.465,-24.353,21.415,-41.558
C09749=1019.518,127.926,366.499,-24.352,21.414,-41.561
C09750=1019.518,127.591,366.533,-24.352,21.415,-41.563
C09751=1019.520,127.257,366.566,-24.352,21.415,-41.565
C09752=1019.521,126.923,366.600,-24.351,21.415,-41.569
C09753=1019.522,126.589,366.635,-24.351,21.415,-41.571
C09754=1019.523,126.256,366.668,-24.351,21.416,-41.572
C09755=1019.525,125.922,366.701,-24.350,21.415,-41.576
C09756=1019.526,125.587,366.735,-24.350,21.416,-41.578
C09757=1019.527,125.253,366.768,-24.349,21.416,-41.581
C09758=1019.529,124.920,366.803,-24.349,21.416,-41.583
C09759=1019.529,124.586,366.837,-24.349,21.416,-41.585
C09760=1019.531,124.252,366.870,-24.348,21.417,-41.589
C09761=1019.532,123.918,366.904,-24.348,21.417,-41.591
C09762=1019.534,123.583,366.938,-24.348,21.417,-41.594
C09763=1019.535,123.249,366.971,-24.347,21.417,-41.596
C09764=1019.536,122.916,367.005,-24.347,21.418,-41.598
C09765=1019.537,122.581,367.039,-24.347,21.418,-41.602
C09766=1019.538,122.248,367.072,-24.346,21.418,-41.604
C09767=1019.539,121.914,367.106,-24.346,21.417,-41.607
C09768=1019.541,121.580,367.139,-24.346,21.418,-41.609
C09769=1019.542,121.246,367.173,-24.345,21.418,-41.613
C09770=1019.544,120.912,367.207,-24.345,21.418,-41.614
C09771=1019.545,120.578,367.240,-24.345,21.419,-41.617
C09772=1019.546,120.244,367.273,-24.344,21.419,-41.620
C09773=1019.547,119.910,367.307,-24.344,21.419,-41.622
C09774=1019.548,119.576,367.341,-24.343,21.419,-41.625
C09775=1019.550,119.243,367.375,-24.343,21.420,-41.628
C09776=1019.551,118.909,367.408,-24.342,21.419,-41.631
C09777=1019.552,118.574,367.442,-24.342,21.420,-41.633
C09778=1019.553,118.240,367.475,-24.342,21.421,-41.635
C09779=1019.554,117.907,367.508,-24.341,21.420,-41.638
C09780=1019.556,117.573,367.542,-24.341,21.421,-41.640
C09781=1019.557,117.238,367.576,-24.341,21.421,-41.644
C09782=1019.558,116.904,367.609,-24.340,21.421,-41.646
C09783=1019.559,116.571,367.642,-24.340,21.421,-41.649
C09784=1019.560,116.237,367.675,-24.340,21.422,-41.652
C09785=1019.562,115.903,367.709,-24.339,21.422,-41.655
C09786=1019.563,115.569,367.743,-24.339,21.422,-41.657
C09787=1019.564,115.235,367.776,-24.338,21.421,-41.660
C09788=1019.565,114.901,367.809,-24.338,21.422,-41.662
C09789=1019.568,114.566,367.842,-24.338,21.423,-41.664
C09790=1019.569,114.233,367.876,-24.337,21.422,-41.668
C09791=1019.570,113.899,367.909,-24.337,21.423,-41.670
C09792=1019.570,113.565,367.942,-24.336,21.423,-41.673
C09793=1019.572,113.231,367.976,-24.336,21.423,-41.675
C09794=1019.573,112.897,368.009,-24.336,21.424,-41.679
C09795=1019.575,112.563,368.043,-24.335,21.424,-41.681
C09796=1019.576,112.229,368.076,-24.335,21.423,-41.684
C09797=1019.576,111.895,368.109,-24.335,21.425,-41.686
C09798=1019.578,111.561,368.143,-24.334,21.424,-41.690
C09799=1019.579,111.227,368.175,-24.334,21.424,-41.692
C09800=1019.580,110.893,368.208,-24.333,21.425,-41.695
C09801=1019.581,110.559,368.242,-24.333,21.425,-41.697
C09802=1019.583,110.226,368.275,-24.333,21.425,-41.701
C09803=1019.585,109.892,368.309,-24.332,21.426,-41.703
C09804=1019.585,109.557,368.342,-24.332,21.425,-41.706
C09805=1019.587,109.223,368.375,-24.332,21.426,-41.708
C09806=1019.588,108.889,368.408,-24.331,21.426,-41.712
C09807=1019.589,108.556,368.441,-24.331,21.426,-41.714
C09808=1019.590,108.222,368.474,-24.330,21.427,-41.718
C09809=1019.592,107.887,368.507,-24.330,21.427,-41.719
C09810=1019.592,107.553,368.540,-24.329,21.427,-41.723
C09811=1019.593,107.219,368.574,-24.329,21.428,-41.725
C09812=1019.595,106.885,368.606,-24.329,21.427,-41.728
C09813=1019.596,106.551,368.639,-24.328,21.427,-41.730
C09814=1019.597,106.218,368.673,-24.328,21.428,-41.734
C09815=1019.598,105.884,368.706,-24.328,21.428,-41.736
C09816=1019.599,105.549,368.739,-24.327,21.428,-41.739
C09817=1019.601,105.215,368.772,-24.327,21.429,-41.742
C09818=1019.602,104.881,368.804,-24.326,21.428,-41.745
C09819=1019.603,104.547,368.838,-24.326,21.430,-41.747
C09820=1019.604,104.213,368.871,-24.326,21.429,-41.751
C09821=1019.606,103.879,368.903,-24.325,21.429,-41.752
C09822=1019.607,103.545,368.937,-24.325,21.430,-41.756
C09823=1019.608,103.211,368.970,-24.324,21.429,-41.760
C09824=1019.609,102.876,369.003,-24.324,21.431,-41.762
C09825=1019.610,102.543,369.036,-24.324,21.430,-41.765
C09826=1019.612,102.208,369.068,-24.323,21.430,-41.767
C09827=1019.613,101.875,369.102,-24.323,21.431,-41.771
C09828=1019.614,101.540,369.134,-24.323,21.431,-41.773
C09829=1019.615,101.206,369.168,-24.322,21.431,-41.776
C09830=1019.616,100.871,369.200,-24.322,21.432,-41.778
C09831=1019.618,100.538,369.233,-24.321,21.431,-41.782
C09832=1019.619,100.203,369.266,-24.321,21.432,-41.785
C09833=1019.620,99.870,369.299,-24.320,21.432,-41.787
C09834=1019.620,99.535,369.331,-24.320,21.432,-41.791
C09835=1019.622,99.201,369.365,-24.320,21.433,-41.793
C09836=1019.623,98.867,369.397,-24.319,21.432,-41.796
C09837=1019.625,98.533,369.430,-24.319,21.433,-41.799
C09838=1019.626,98.199,369.463,-24.318,21.433,-41.802
C09839=1019.627,97.864,369.495,-24.318,21.433,-41.806
C09840=1019.628,97.530,369.529,-24.318,21.434,-41.808
C09841=1019.629,97.196,369.561,-24.317,21.434,-41.811
C09842=1019.630,96.862,369.593,-24.317,21.434,-41.813
C09843=1019.631,96.528,369.627,-24.316,21.434,-41.817
C09844=1019.632,96.193,369.659,-24.316,21.435,-41.819
C09845=1019.634,95.859,369.692,-24.316,21.435,-41.822
C09846=1019.635,95.524,369.725,-24.315,21.435,-41.826
C09847=1019.636,95.190,369.758,-24.315,21.435,-41.828
C09848=1019.638,94.856,369.790,-24.314,21.436,-41.832
C09849=1019.638,94.521,369.823,-24.314,21.436,-41.833
C09850=1019.639,94.187,369.855,-24.314,21.436,-41.837
C09851=1019.641,93.853,369.888,-24.313,21.436,-41.841
C09852=1019.642,93.519,369.921,-24.313,21.436,-41.842
C09853=1019.643,93.184,369.954,-24.312,21.437,-41.846
C09854=1019.644,92.850,369.986,-24.312,21.436,-41.849
C09855=1019.645,92.516,370.018,-24.311,21.437,-41.852
C09856=1019.646,92.181,370.052,-24.311,21.437,-41.855
C09857=1019.647,91.847,370.084,-24.311,21.438,-41.857
C09858=1019.649,91.512,370.117,-24.310,21.438,-41.861
C09859=1019.650,91.178,370.149,-24.310,21.438,-41.865
C09860=1019.650,90.843,370.181,-24.309,21.438,-41.866
C09861=1019.652,90.509,370.214,-24.309,21.439,-41.870
C09862=1019.653,90.175,370.246,-24.308,21.438,-41.874
C09863=1019.654,89.841,370.279,-24.308,21.440,-41.876
C09864=1019.655,89.512,370.311,-24.308,21.439,-41.879
C09865=1019.656,89.187,370.342,-24.307,21.439,-41.881
C09866=1019.657,88.866,370.374,-24.307,21.440,-41.885
C09867=1019.658,88.546,370.405,-24.306,21.439,-41.888
C09868=1019.659,88.223,370.436,-24.306,21.441,-41.890
C09869=1019.660,87.897,370.468,-24.305,21.440,-41.894
C09870=1019.661,87.564,370.500,-24.305,21.441,-41.898
C09871=1019.662,87.228,370.532,-24.305,21.441,-41.899
C09872=1019.664,86.888,370.566,-24.304,21.441,-41.903
C09873=1019.665,86.547,370.598,-24.304,21.441,-41.906
C09874=1019.665,86.205,370.631,-24.303,21.442,-41.909
C09875=1019.667,85.863,370.664,-24.303,21.442,-41.912
C09876=1019.668,85.518,370.698,-24.302,21.442,-41.916
C09877=1019.669,85.173,370.731,-24.302,21.443,-41.918
C09878=1019.670,84.826,370.764,-24.302,21.443,-41.922
C09879=1019.671,84.478,370.798,-24.301,21.443,-41.925
C09880=1019.672,84.130,370.832,-24.301,21.443,-41.929
C09881=1019.674,83.779,370.866,-24.300,21.444,-41.931
C09882=1019.675,83.429,370.900,-24.300,21.444,-41.935
C09883=1019.676,83.077,370.933,-24.299,21.444,-41.938
C09884=1019.677,82.724,370.967,-24.299,21.444,-41.942
C09885=1019.678,82.370,371.001,-24.298,21.444,-41.945
C09886=1019.679,82.016,371.036,-24.298,21.445,-41.947
C09887=1019.680,81.660,371.070,-24.298,21.446,-41.951
C09888=1019.682,81.304,371.104,-24.297,21.445,-41.955
C09889=1019.682,80.948,371.138,-24.297,21.446,-41.958
C09890=1019.683,80.591,371.173,-24.296,21.446,-41.962
C09891=1019.685,80.236,371.207,-24.296,21.446,-41.964
C09892=1019.686,79.885,371.240,-24.295,21.447,-41.968
C09893=1019.687,79.539,371.274,-24.295,21.446,-41.971
C09894=1019.688,79.201,371.306,-24.295,21.448,-41.973
C09895=1019.690,78.868,371.338,-24.294,21.447,-41.977
C09896=1019.690,78.540,371.370,-24.293,21.448,-41.980
C09897=1019.690,78.215,371.401,-24.293,21.448,-41.984
C09898=1019.693,77.892,371.432,-24.292,21.448,-41.987
C09899=1019.693,77.568,371.463,-24.292,21.449,-41.990
C09900=1019.694,77.242,371.494,-24.292,21.449,-41.994
C09901=1019.695,76.912,371.525,-24.291,21.449,-41.997
C09902=1019.696,76.576,371.557,-24.291,21.449,-42.001
C09903=1019.697,76.234,371.590,-24.290,21.449,-42.004
C09904=1019.698,75.885,371.624,-24.290,21.450,-42.006
C09905=1019.700,75.532,371.658,-24.289,21.450,-42.010
C09906=1019.699,75.174,371.691,-24.289,21.450,-42.013
C09907=1019.702,74.816,371.726,-24.288,21.451,-42.017
C09908=1019.702,74.459,371.759,-24.288,21.451,-42.019
C09909=1019.703,74.104,371.793,-24.288,21.451,-42.023
C09910=1019.705,73.750,371.827,-24.287,21.452,-42.027
C09911=1019.705,73.399,371.860,-24.286,21.451,-42.030
C09912=1019.706,73.049,371.893,-24.286,21.452,-42.034
C09913=1019.708,72.701,371.927,-24.285,21.452,-42.037
C09914=1019.709,72.355,371.959,-24.285,21.453,-42.041
C09915=1019.709,72.009,371.993,-24.285,21.453,-42.043
C09916=1019.711,71.664,372.025,-24.284,21.453,-42.047
C09917=1019.712,71.320,372.058,-24.284,21.454,-42.051
C09918=1019.712,70.976,372.092,-24.283,21.453,-42.054
C09919=1019.714,70.631,372.123,-24.283,21.454,-42.058
C09920=1019.715,70.286,372.156,-24.282,21.454,-42.061
C09921=1019.716,69.942,372.189,-24.282,21.455,-42.063
C09922=1019.716,69.598,372.221,-24.281,21.455,-42.067
C09923=1019.718,69.255,372.254,-24.281,21.456,-42.071
C09924=1019.719,68.913,372.286,-24.280,21.455,-42.074
C09925=1019.719,68.572,372.319,-24.280,21.456,-42.078
C09926=1019.721,68.232,372.351,-24.279,21.456,-42.082
C09927=1019.722,67.892,372.383,-24.279,21.456,-42.085
C09928=1019.722,67.554,372.415,-24.279,21.457,-42.087
C09929=1019.723,67.217,372.447,-24.278,21.457,-42.091
C09930=1019.724,66.880,372.478,-24.278,21.457,-42.094
C09931=1019.725,66.544,372.510,-24.277,21.457,-42.098
C09932=1019.726,66.211,372.541,-24.277,21.458,-42.102
C09933=1019.727,65.872,372.574,-24.276,21.457,-42.105
C09934=1019.728,65.518,372.606,-24.276,21.459,-42.108
C09935=1019.729,65.141,372.643,-24.275,21.458,-42.113
C09936=1019.730,64.745,372.680,-24.274,21.459,-42.116
C09937=1019.732,64.359,372.716,-24.274,21.459,-42.120
C09938=1019.732,64.004,372.750,-24.274,21.460,-42.124
C09939=1019.733,63.629,372.785,-24.273,21.460,-42.128
C09940=1019.734,63.411,372.805,-24.273,21.461,-42.130
C09941=1019.735,63.187,372.826,-24.272,21.460,-42.131
C09942=1019.740,62.792,372.860,-24.272,21.460,-42.135
C09943=1019.744,62.456,372.890,-24.271,21.461,-42.139
C09944=1019.749,62.120,372.920,-24.271,21.461,-42.142
C09945=1019.753,61.785,372.949,-24.270,21.462,-42.146
C09946=1019.757,61.450,372.978,-24.270,21.461,-42.149
C09947=1019.761,61.114,373.008,-24.269,21.462,-42.153
C09948=1019.765,60.780,373.038,-24.269,21.462,-42.157
C09949=1019.768,60.444,373.067,-24.268,21.462,-42.160
C09950=1019.773,60.110,373.096,-24.268,21.463,-42.163
C09951=1019.776,59.775,373.126,-24.268,21.464,-42.166
C09952=1019.781,59.440,373.155,-24.267,21.464,-42.170
C09953=1019.785,59.105,373.185,-24.267,21.464,-42.173
C09954=1019.788,58.769,373.214,-24.266,21.464,-42.177
C09955=1019.792,58.434,373.243,-24.266,21.465,-42.181
C09956=1019.796,58.100,373.273,-24.265,21.464,-42.184
C09957=1019.800,57.764,373.302,-24.264,21.465,-42.188
C09958=1019.804,57.429,373.332,-24.264,21.465,-42.192
C09959=1019.808,57.094,373.361,-24.264,21.466,-42.194
C09960=1019.812,56.760,373.390,-24.263,21.466,-42.197
C09961=1019.816,56.425,373.420,-24.263,21.466,-42.201
C09962=1019.820,56.089,373.449,-24.262,21.467,-42.205
C09963=1019.823,55.755,373.479,-24.262,21.467,-42.209
C09964=1019.827,55.419,373.507,-24.261,21.467,-42.212
C09965=1019.831,55.084,373.537,-24.261,21.467,-42.216
C09966=1019.834,54.750,373.567,-24.260,21.468,-42.220
C09967=1019.838,54.414,373.596,-24.260,21.468,-42.223
C09968=1019.842,54.079,373.625,-24.259,21.468,-42.227
C09969=1019.846,53.744,373.654,-24.259,21.468,-42.230
C09970=1019.849,53.409,373.684,-24.258,21.469,-42.234
C09971=1019.853,53.074,373.713,-24.258,21.469,-42.238
C09972=1019.857,52.739,373.742,-24.257,21.470,-42.240
C09973=1019.860,52.404,373.772,-24.257,21.470,-42.244
C09974=1019.864,52.069,373.800,-24.256,21.470,-42.247
C09975=1019.867,51.734,373.830,-24.256,21.471,-42.251
C09976=1019.871,51.399,373.859,-24.255,21.471,-42.254
C09977=1019.875,51.050,373.889,-24.255,21.471,-42.258
C09978=1020.027,-120.097,387.201,-23.946,21.709,-44.569
C09979=1020.024,-120.382,387.220,-23.945,21.709,-44.573
C09980=1020.022,-120.666,387.240,-23.945,21.710,-44.577
C09981=1020.018,-120.995,387.262,-23.944,21.710,-44.582
C09982=1020.014,-121.323,387.284,-23.944,21.711,-44.586
C09983=1020.011,-121.651,387.305,-23.943,21.711,-44.591
C09984=1020.008,-121.980,387.328,-23.942,21.712,-44.597
C09985=1020.005,-122.308,387.350,-23.942,21.713,-44.601
C09986=1020.001,-122.636,387.372,-23.941,21.713,-44.606
C09987=1019.998,-122.964,387.394,-23.940,21.714,-44.610
C09988=1019.995,-123.292,387.417,-23.940,21.714,-44.615
C09989=1019.991,-123.621,387.438,-23.939,21.715,-44.620
C09990=1019.988,-123.949,387.460,-23.939,21.715,-44.625
C09991=1019.984,-124.277,387.482,-23.938,21.716,-44.628
C09992=1019.980,-124.605,387.504,-23.937,21.717,-44.634
//INST
///DATE 2021/06/25 14:57
///ATTR SC,RW,RJ
////FRAME ROBOT
///GROUP1 RB1
NOP
MOVL C00000 V=800.0 PL=0
MOVL C00001 V=800.0 PL=0
MOVL C00002 V=800.0 PL=0
MOVL C00003 V=800.0 PL=0
MOVL C00004 V=800.0 PL=0
MOVL C00005 V=800.0 PL=0
MOVL C00006 V=800.0 PL=0
MOVL C00007 V=800.0 PL=0
MOVL C00008 V=800.0 PL=0
MOVL C00009 V=800.0 PL=0
MOVL C00010 V=800.0 PL=0
MOVL C00011 V=800.0 PL=0
MOVL C00012 V=800.0 PL=0
MOVL C00013 V=800.0 PL=0
MOVL C00014 V=800.0 PL=0
MOVL C00015 V=800.0 PL=0
MOVL C00016 V=800.0 PL=0
MOVL C00017 V=800.0 PL=0
MOVL C00018 V=800.0 PL=0
MOVL C00019 V=800.0 PL=0
MOVL C00020 V=800.0 PL=0
MOVL C00021 V=800.0 PL=0
MOVL C00022 V=800.0 PL=0
MOVL C00023 V=800.0 PL=0
MOVL C00024 V=800.0 PL=0
MOVL C00025 V=800.0 PL=0
MOVL C00026 V=800.0 PL=0
MOVL C00027 V=800.0 PL=0
MOVL C00028 V=800.0 PL=0
MOVL C00029 V=800.0 PL=0
MOVL C00030 V=800.0 PL=0
MOVL C00031 V=800.0 PL=0
MOVL C00032 V=800.0 PL=0
MOVL C00033 V=800.0 PL=0
MOVL C00034 V=800.0 PL=0
MOVL C00035 V=800.0 PL=0
MOVL C00036 V=800.0 PL=0
MOVL C00037 V=800.0 PL=0
MOVL C00038 V=800.0 PL=0
MOVL C00039 V=800.0 PL=0
MOVL C00040 V=800.0 PL=0
MOVL C00041 V=800.0 PL=0
MOVL C00042 V=800.0 PL=0
MOVL C00043 V=800.0 PL=0
MOVL C00044 V=800.0 PL=0
MOVL C00045 V=800.0 PL=0
MOVL C00046 V=800.0 PL=0
MOVL C00047 V=800.0 PL=0
MOVL C00048 V=800.0 PL=0
MOVL C00049 V=800.0 PL=0
MOVL C00050 V=800.0 PL=0
MOVL C00051 V=800.0 PL=0
MOVL C00052 V=800.0 PL=0
MOVL C00053 V=800.0 PL=0
MOVL C00054 V=800.0 PL=0
MOVL C00055 V=800.0 PL=0
MOVL C00056 V=800.0 PL=0
MOVL C00057 V=800.0 PL=0
MOVL C00058 V=800.0 PL=0
MOVL C00059 V=800.0 PL=0
MOVL C00060 V=800.0 PL=0
MOVL C00061 V=800.0 PL=0
MOVL C00062 V=800.0 PL=0
MOVL C00063 V=800.0 PL=0
MOVL C00064 V=800.0 PL=0
MOVL C00065 V=800.0 PL=0
MOVL C00066 V=800.0 PL=0
MOVL C00067 V=800.0 PL=0
MOVL C00068 V=800.0 PL=0
MOVL C00069 V=800.0 PL=0
MOVL C00070 V=800.0 PL=0
MOVL C00071 V=800.0 PL=0
MOVL C00072 V=800.0 PL=0
MOVL C00073 V=800.0 PL=0
MOVL C00074 V=800.0 PL=0
MOVL C00075 V=800.0 PL=0
MOVL C00076 V=800.0 PL=0
MOVL C00077 V=800.0 PL=0
MOVL C00078 V=800.0 PL=0
MOVL C00079 V=800.0 PL=0
MOVL C00080 V=800.0 PL=0
MOVL C00081 V=800.0 PL=0
MOVL C00082 V=800.0 PL=0
MOVL C00083 V=800.0 PL=0
MOVL C00084 V=800.0 PL=0
MOVL C00085 V=800.0 PL=0
MOVL C00086 V=800.0 PL=0
MOVL C00087 V=800.0 PL=0
MOVL C00088 V=800.0 PL=0
MOVL C00089 V=800.0 PL=0
MOVL C00090 V=800.0 PL=0
MOVL C00091 V=800.0 PL=0
MOVL C00092 V=800.0 PL=0
MOVL C00093 V=800.0 PL=0
MOVL C00094 V=800.0 PL=0
MOVL C00095 V=800.0 PL=0
MOVL C00096 V=800.0 PL=0
MOVL C00097 V=800.0 PL=0
MOVL C00098 V=800.0 PL=0
MOVL C00099 V=800.0 PL=0
MOVL C00100 V=800.0 PL=0
MOVL C00101 V=800.0 PL=0
MOVL C00102 V=800.0 PL=0
MOVL C00103 V=800.0 PL=0
MOVL C00104 V=800.0 PL=0
MOVL C00105 V=800.0 PL=0
MOVL C00106 V=800.0 PL=0
MOVL C00107 V=800.0 PL=0
MOVL C00108 V=800.0 PL=0
MOVL C00109 V=800.0 PL=0
MOVL C00110 V=800.0 PL=0
MOVL C00111 V=800.0 PL=0
MOVL C00112 V=800.0 PL=0
MOVL C00113 V=800.0 PL=0
MOVL C00114 V=800.0 PL=0
MOVL C00115 V=800.0 PL=0
MOVL C00116 V=800.0 PL=0
MOVL C00117 V=800.0 PL=0
MOVL C00118 V=800.0 PL=0
MOVL C00119 V=800.0 PL=0
MOVL C00120 V=800.0 PL=0
MOVL C00121 V=800.0 PL=0
MOVL C00122 V=800.0 PL=0
MOVL C00123 V=800.0 PL=0
MOVL C00124 V=800.0 PL=0
MOVL C00125 V=800.0 PL=0
MOVL C00126 V=800.0 PL=0
MOVL C00127 V=800.0 PL=0
MOVL C00128 V=800.0 PL=0
MOVL C00129 V=800.0 PL=0
MOVL C00130 V=800.0 PL=0
MOVL C00131 V=800.0 PL=0
MOVL C00132 V=800.0 PL=0
MOVL C00133 V=800.0 PL=0
MOVL C00134 V=800.0 PL=0
MOVL C00135 V=800.0 PL=0
MOVL C00136 V=800.0 PL=0
MOVL C00137 V=800.0 PL=0
MOVL C00138 V=800.0 PL=0
MOVL C00139 V=800.0 PL=0
MOVL C00140 V=800.0 PL=0
MOVL C00141 V=800.0 PL=0
MOVL C00142 V=800.0 PL=0
MOVL C00143 V=800.0 PL=0
MOVL C00144 V=800.0 PL=0
MOVL C00145 V=800.0 PL=0
MOVL C00146 V=800.0 PL=0
MOVL C00147 V=800.0 PL=0
MOVL C00148 V=800.0 PL=0
MOVL C00149 V=800.0 PL=0
MOVL C00150 V=800.0 PL=0
MOVL C00151 V=800.0 PL=0
MOVL C00152 V=800.0 PL=0
MOVL C00153 V=800.0 PL=0
MOVL C00154 V=800.0 PL=0
MOVL C00155 V=800.0 PL=0
MOVL C00156 V=800.0 PL=0
MOVL C00157 V=800.0 PL=0
MOVL C00158 V=800.0 PL=0
MOVL C00159 V=800.0 PL=0
MOVL C00160 V=800.0 PL=0
MOVL C00161 V=800.0 PL=0
MOVL C00162 V=800.0 PL=0
MOVL C00163 V=800.0 PL=0
MOVL C00164 V=800.0 PL=0
MOVL C00165 V=800.0 PL=0
MOVL C00166 V=800.0 PL=0
MOVL C00167 V=800.0 PL=0
MOVL C00168 V=800.0 PL=0
MOVL C00169 V=800.0 PL=0
MOVL C00170 V=800.0 PL=0
MOVL C00171 V=800.0 PL=0
MOVL C00172 V=800.0 PL=0
MOVL C00173 V=800.0 PL=0
MOVL C00174 V=800.0 PL=0
MOVL C00175 V=800.0 PL=0
MOVL C00176 V=800.0 PL=0
MOVL C00177 V=800.0 PL=0
MOVL C00178 V=800.0 PL=0
MOVL C00179 V=800.0 PL=0
MOVL C00180 V=800.0 PL=0
MOVL C00181 V=800.0 PL=0
MOVL C00182 V=800.0 PL=0
MOVL C00183 V=800.0 PL=0
MOVL C00184 V=800.0 PL=0
MOVL C00185 V=800.0 PL=0
MOVL C00186 V=800.0 PL=0
MOVL C00187 V=800.0 PL=0
MOVL C00188 V=800.0 PL=0
MOVL C00189 V=800.0 PL=0
MOVL C00190 V=800.0 PL=0
MOVL C00191 V=800.0 PL=0
MOVL C00192 V=800.0 PL=0
MOVL C00193 V=800.0 PL=0
MOVL C00194 V=800.0 PL=0
MOVL C00195 V=800.0 PL=0
MOVL C00196 V=800.0 PL=0
MOVL C00197 V=800.0 PL=0
MOVL C00198 V=800.0 PL=0
MOVL C00199 V=800.0 PL=0
MOVL C00200 V=800.0 PL=0
MOVL C00201 V=800.0 PL=0
MOVL C00202 V=800.0 PL=0
MOVL C00203 V=800.0 PL=0
MOVL C00204 V=800.0 PL=0
MOVL C00205 V=800.0 PL=0
MOVL C00206 V=800.0 PL=0
MOVL C00207 V=800.0 PL=0
MOVL C00208 V=800.0 PL=0
MOVL C00209 V=800.0 PL=0
MOVL C00210 V=800.0 PL=0
MOVL C00211 V=800.0 PL=0
MOVL C00212 V=800.0 PL=0
MOVL C00213 V=800.0 PL=0
MOVL C00214 V=800.0 PL=0
MOVL C00215 V=800.0 PL=0
MOVL C00216 V=800.0 PL=0
MOVL C00217 V=800.0 PL=0
MOVL C00218 V=800.0 PL=0
MOVL C00219 V=800.0 PL=0
MOVL C00220 V=800.0 PL=0
MOVL C00221 V=800.0 PL=0
MOVL C00222 V=800.0 PL=0
MOVL C00223 V=800.0 PL=0
MOVL C00224 V=800.0 PL=0
MOVL C00225 V=800.0 PL=0
MOVL C00226 V=800.0 PL=0
MOVL C00227 V=800.0 PL=0
MOVL C00228 V=800.0 PL=0
MOVL C00229 V=800.0 PL=0
MOVL C00230 V=800.0 PL=0
MOVL C00231 V=800.0 PL=0
MOVL C00232 V=800.0 PL=0
MOVL C00233 V=800.0 PL=0
MOVL C00234 V=800.0 PL=0
MOVL C00235 V=800.0 PL=0
MOVL C00236 V=800.0 PL=0
MOVL C00237 V=800.0 PL=0
MOVL C00238 V=800.0 PL=0
MOVL C00239 V=800.0 PL=0
MOVL C00240 V=800.0 PL=0
MOVL C00241 V=800.0 PL=0
MOVL C00242 V=800.0 PL=0
MOVL C00243 V=800.0 PL=0
MOVL C00244 V=800.0 PL=0
MOVL C00245 V=800.0 PL=0
MOVL C00246 V=800.0 PL=0
MOVL C00247 V=800.0 PL=0
MOVL C00248 V=800.0 PL=0
MOVL C00249 V=800.0 PL=0
MOVL C00250 V=800.0 PL=0
MOVL C00251 V=800.0 PL=0
MOVL C00252 V=800.0 PL=0
MOVL C00253 V=800.0 PL=0
MOVL C00254 V=800.0 PL=0
MOVL C00255 V=800.0 PL=0
MOVL C00256 V=800.0 PL=0
MOVL C00257 V=800.0 PL=0
MOVL C00258 V=800.0 PL=0
MOVL C00259 V=800.0 PL=0
MOVL C00260 V=800.0 PL=0
MOVL C00261 V=800.0 PL=0
MOVL C00262 V=800.0 PL=0
MOVL C00263 V=800.0 PL=0
MOVL C00264 V=800.0 PL=0
MOVL C00265 V=800.0 PL=0
MOVL C00266 V=800.0 PL=0
MOVL C00267 V=800.0 PL=0
MOVL C00268 V=800.0 PL=0
MOVL C00269 V=800.0 PL=0
MOVL C00270 V=800.0 PL=0
MOVL C00271 V=800.0 PL=0
MOVL C00272 V=800.0 PL=0
MOVL C00273 V=800.0 PL=0
MOVL C00274 V=800.0 PL=0
MOVL C00275 V=800.0 PL=0
MOVL C00276 V=800.0 PL=0
MOVL C00277 V=800.0 PL=0
MOVL C00278 V=800.0 PL=0
MOVL C00279 V=800.0 PL=0
MOVL C00280 V=800.0 PL=0
MOVL C00281 V=800.0 PL=0
MOVL C00282 V=800.0 PL=0
MOVL C00283 V=800.0 PL=0
MOVL C00284 V=800.0 PL=0
MOVL C00285 V=800.0 PL=0
MOVL C00286 V=800.0 PL=0
MOVL C00287 V=800.0 PL=0
MOVL C00288 V=800.0 PL=0
MOVL C00289 V=800.0 PL=0
MOVL C00290 V=800.0 PL=0
MOVL C00291 V=800.0 PL=0
MOVL C00292 V=800.0 PL=0
MOVL C00293 V=800.0 PL=0
MOVL C00294 V=800.0 PL=0
MOVL C00295 V=800.0 PL=0
MOVL C00296 V=800.0 PL=0
MOVL C00297 V=800.0 PL=0
MOVL C00298 V=800.0 PL=0
MOVL C00299 V=800.0 PL=0
MOVL C00300 V=800.0 PL=0
MOVL C00301 V=800.0 PL=0
MOVL C00302 V=800.0 PL=0
MOVL C00303 V=800.0 PL=0
MOVL C00304 V=800.0 PL=0
MOVL C00305 V=800.0 PL=0
MOVL C00306 V=800.0 PL=0
MOVL C00307 V=800.0 PL=0
MOVL C00308 V=800.0 PL=0
MOVL C00309 V=800.0 PL=0
MOVL C00310 V=800.0 PL=0
MOVL C00311 V=800.0 PL=0
MOVL C00312 V=800.0 PL=0
MOVL C00313 V=800.0 PL=0
MOVL C00314 V=800.0 PL=0
MOVL C00315 V=800.0 PL=0
MOVL C00316 V=800.0 PL=0
MOVL C00317 V=800.0 PL=0
MOVL C00318 V=800.0 PL=0
MOVL C00319 V=800.0 PL=0
MOVL C00320 V=800.0 PL=0
MOVL C00321 V=800.0 PL=0
MOVL C00322 V=800.0 PL=0
MOVL C00323 V=800.0 PL=0
MOVL C00324 V=800.0 PL=0
MOVL C00325 V=800.0 PL=0
MOVL C00326 V=800.0 PL=0
MOVL C00327 V=800.0 PL=0
MOVL C00328 V=800.0 PL=0
MOVL C00329 V=800.0 PL=0
MOVL C00330 V=800.0 PL=0
MOVL C00331 V=800.0 PL=0
MOVL C00332 V=800.0 PL=0
MOVL C00333 V=800.0 PL=0
MOVL C00334 V=800.0 PL=0
MOVL C00335 V=800.0 PL=0
MOVL C00336 V=800.0 PL=0
MOVL C00337 V=800.0 PL=0
MOVL C00338 V=800.0 PL=0
MOVL C00339 V=800.0 PL=0
MOVL C00340 V=800.0 PL=0
MOVL C00341 V=800.0 PL=0
MOVL C00342 V=800.0 PL=0
MOVL C00343 V=800.0 PL=0
MOVL C00344 V=800.0 PL=0
MOVL C00345 V=800.0 PL=0
MOVL C00346 V=800.0 PL=0
MOVL C00347 V=800.0 PL=0
MOVL C00348 V=800.0 PL=0
MOVL C00349 V=800.0 PL=0
MOVL C00350 V=800.0 PL=0
MOVL C00351 V=800.0 PL=0
MOVL C00352 V=800.0 PL=0
MOVL C00353 V=800.0 PL=0
MOVL C00354 V=800.0 PL=0
MOVL C00355 V=800.0 PL=0
MOVL C00356 V=800.0 PL=0
MOVL C00357 V=800.0 PL=0
MOVL C00358 V=800.0 PL=0
MOVL C00359 V=800.0 PL=0
MOVL C00360 V=800.0 PL=0
MOVL C00361 V=800.0 PL=0
MOVL C00362 V=800.0 PL=0
MOVL C00363 V=800.0 PL=0
MOVL C00364 V=800.0 PL=0
MOVL C00365 V=800.0 PL=0
MOVL C00366 V=800.0 PL=0
MOVL C00367 V=800.0 PL=0
MOVL C00368 V=800.0 PL=0
MOVL C00369 V=800.0 PL=0
MOVL C00370 V=800.0 PL=0
MOVL C00371 V=800.0 PL=0
MOVL C00372 V=800.0 PL=0
MOVL C00373 V=800.0 PL=0
MOVL C00374 V=800.0 PL=0
MOVL C00375 V=800.0 PL=0
MOVL C00376 V=800.0 PL=0
MOVL C00377 V=800.0 PL=0
MOVL C00378 V=800.0 PL=0
MOVL C00379 V=800.0 PL=0
MOVL C00380 V=800.0 PL=0
MOVL C00381 V=800.0 PL=0
MOVL C00382 V=800.0 PL=0
MOVL C00383 V=800.0 PL=0
MOVL C00384 V=800.0 PL=0
MOVL C00385 V=800.0 PL=0
MOVL C00386 V=800.0 PL=0
MOVL C00387 V=800.0 PL=0
MOVL C00388 V=800.0 PL=0
MOVL C00389 V=800.0 PL=0
MOVL C00390 V=800.0 PL=0
MOVL C00391 V=800.0 PL=0
MOVL C00392 V=800.0 PL=0
MOVL C00393 V=800.0 PL=0
MOVL C00394 V=800.0 PL=0
MOVL C00395 V=800.0 PL=0
MOVL C00396 V=800.0 PL=0
MOVL C00397 V=800.0 PL=0
MOVL C00398 V=800.0 PL=0
MOVL C00399 V=800.0 PL=0
MOVL C00400 V=800.0 PL=0
MOVL C00401 V=800.0 PL=0
MOVL C00402 V=800.0 PL=0
MOVL C00403 V=800.0 PL=0
MOVL C00404 V=800.0 PL=0
MOVL C00405 V=800.0 PL=0
MOVL C00406 V=800.0 PL=0
MOVL C00407 V=800.0 PL=0
MOVL C00408 V=800.0 PL=0
MOVL C00409 V=800.0 PL=0
MOVL C00410 V=800.0 PL=0
MOVL C00411 V=800.0 PL=0
MOVL C00412 V=800.0 PL=0
MOVL C00413 V=800.0 PL=0
MOVL C00414 V=800.0 PL=0
MOVL C00415 V=800.0 PL=0
MOVL C00416 V=800.0 PL=0
MOVL C00417 V=800.0 PL=0
MOVL C00418 V=800.0 PL=0
MOVL C00419 V=800.0 PL=0
MOVL C00420 V=800.0 PL=0
MOVL C00421 V=800.0 PL=0
MOVL C00422 V=800.0 PL=0
MOVL C00423 V=800.0 PL=0
MOVL C00424 V=800.0 PL=0
MOVL C00425 V=800.0 PL=0
MOVL C00426 V=800.0 PL=0
MOVL C00427 V=800.0 PL=0
MOVL C00428 V=800.0 PL=0
MOVL C00429 V=800.0 PL=0
MOVL C00430 V=800.0 PL=0
MOVL C00431 V=800.0 PL=0
MOVL C00432 V=800.0 PL=0
MOVL C00433 V=800.0 PL=0
MOVL C00434 V=800.0 PL=0
MOVL C00435 V=800.0 PL=0
MOVL C00436 V=800.0 PL=0
MOVL C00437 V=800.0 PL=0
MOVL C00438 V=800.0 PL=0
MOVL C00439 V=800.0 PL=0
MOVL C00440 V=800.0 PL=0
MOVL C00441 V=800.0 PL=0
MOVL C00442 V=800.0 PL=0
MOVL C00443 V=800.0 PL=0
MOVL C00444 V=800.0 PL=0
MOVL C00445 V=800.0 PL=0
MOVL C00446 V=800.0 PL=0
MOVL C00447 V=800.0 PL=0
MOVL C00448 V=800.0 PL=0
MOVL C00449 V=800.0 PL=0
MOVL C00450 V=800.0 PL=0
MOVL C00451 V=800.0 PL=0
MOVL C00452 V=800.0 PL=0
MOVL C00453 V=800.0 PL=0
MOVL C00454 V=800.0 PL=0
MOVL C00455 V=800.0 PL=0
MOVL C00456 V=800.0 PL=0
MOVL C00457 V=800.0 PL=0
MOVL C00458 V=800.0 PL=0
MOVL C00459 V=800.0 PL=0
MOVL C00460 V=800.0 PL=0
MOVL C00461 V=800.0 PL=0
MOVL C00462 V=800.0 PL=0
MOVL C00463 V=800.0 PL=0
MOVL C00464 V=800.0 PL=0
MOVL C00465 V=800.0 PL=0
MOVL C00466 V=800.0 PL=0
MOVL C00467 V=800.0 PL=0
MOVL C00468 V=800.0 PL=0
MOVL C00469 V=800.0 PL=0
MOVL C00470 V=800.0 PL=0
MOVL C00471 V=800.0 PL=0
MOVL C00472 V=800.0 PL=0
MOVL C00473 V=800.0 PL=0
MOVL C00474 V=800.0 PL=0
MOVL C00475 V=800.0 PL=0
MOVL C00476 V=800.0 PL=0
MOVL C00477 V=800.0 PL=0
MOVL C00478 V=800.0 PL=0
MOVL C00479 V=800.0 PL=0
MOVL C00480 V=800.0 PL=0
MOVL C00481 V=800.0 PL=0
MOVL C00482 V=800.0 PL=0
MOVL C00483 V=800.0 PL=0
MOVL C00484 V=800.0 PL=0
MOVL C00485 V=800.0 PL=0
MOVL C00486 V=800.0 PL=0
MOVL C00487 V=800.0 PL=0
MOVL C00488 V=800.0 PL=0
MOVL C00489 V=800.0 PL=0
MOVL C00490 V=800.0 PL=0
MOVL C00491 V=800.0 PL=0
MOVL C00492 V=800.0 PL=0
MOVL C00493 V=800.0 PL=0
MOVL C00494 V=800.0 PL=0
MOVL C00495 V=800.0 PL=0
MOVL C00496 V=800.0 PL=0
MOVL C00497 V=800.0 PL=0
MOVL C00498 V=800.0 PL=0
MOVL C00499 V=800.0 PL=0
MOVL C00500 V=800.0 PL=0
MOVL C00501 V=800.0 PL=0
MOVL C00502 V=800.0 PL=0
MOVL C00503 V=800.0 PL=0
MOVL C00504 V=800.0 PL=0
MOVL C00505 V=800.0 PL=0
MOVL C00506 V=800.0 PL=0
MOVL C00507 V=800.0 PL=0
MOVL C00508 V=800.0 PL=0
MOVL C00509 V=800.0 PL=0
MOVL C00510 V=800.0 PL=0
MOVL C00511 V=800.0 PL=0
MOVL C00512 V=800.0 PL=0
MOVL C00513 V=800.0 PL=0
MOVL C00514 V=800.0 PL=0
MOVL C00515 V=800.0 PL=0
MOVL C00516 V=800.0 PL=0
MOVL C00517 V=800.0 PL=0
MOVL C00518 V=800.0 PL=0
MOVL C00519 V=800.0 PL=0
MOVL C00520 V=800.0 PL=0
MOVL C00521 V=800.0 PL=0
MOVL C00522 V=800.0 PL=0
MOVL C00523 V=800.0 PL=0
MOVL C00524 V=800.0 PL=0
MOVL C00525 V=800.0 PL=0
MOVL C00526 V=800.0 PL=0
MOVL C00527 V=800.0 PL=0
MOVL C00528 V=800.0 PL=0
MOVL C00529 V=800.0 PL=0
MOVL C00530 V=800.0 PL=0
MOVL C00531 V=800.0 PL=0
MOVL C00532 V=800.0 PL=0
MOVL C00533 V=800.0 PL=0
MOVL C00534 V=800.0 PL=0
MOVL C00535 V=800.0 PL=0
MOVL C00536 V=800.0 PL=0
MOVL C00537 V=800.0 PL=0
MOVL C00538 V=800.0 PL=0
MOVL C00539 V=800.0 PL=0
MOVL C00540 V=800.0 PL=0
MOVL C00541 V=800.0 PL=0
MOVL C00542 V=800.0 PL=0
MOVL C00543 V=800.0 PL=0
MOVL C00544 V=800.0 PL=0
MOVL C00545 V=800.0 PL=0
MOVL C00546 V=800.0 PL=0
MOVL C00547 V=800.0 PL=0
MOVL C00548 V=800.0 PL=0
MOVL C00549 V=800.0 PL=0
MOVL C00550 V=800.0 PL=0
MOVL C00551 V=800.0 PL=0
MOVL C00552 V=800.0 PL=0
MOVL C00553 V=800.0 PL=0
MOVL C00554 V=800.0 PL=0
MOVL C00555 V=800.0 PL=0
MOVL C00556 V=800.0 PL=0
MOVL C00557 V=800.0 PL=0
MOVL C00558 V=800.0 PL=0
MOVL C00559 V=800.0 PL=0
MOVL C00560 V=800.0 PL=0
MOVL C00561 V=800.0 PL=0
MOVL C00562 V=800.0 PL=0
MOVL C00563 V=800.0 PL=0
MOVL C00564 V=800.0 PL=0
MOVL C00565 V=800.0 PL=0
MOVL C00566 V=800.0 PL=0
MOVL C00567 V=800.0 PL=0
MOVL C00568 V=800.0 PL=0
MOVL C00569 V=800.0 PL=0
MOVL C00570 V=800.0 PL=0
MOVL C00571 V=800.0 PL=0
MOVL C00572 V=800.0 PL=0
MOVL C00573 V=800.0 PL=0
MOVL C00574 V=800.0 PL=0
MOVL C00575 V=800.0 PL=0
MOVL C00576 V=800.0 PL=0
MOVL C00577 V=800.0 PL=0
MOVL C00578 V=800.0 PL=0
MOVL C00579 V=800.0 PL=0
MOVL C00580 V=800.0 PL=0
MOVL C00581 V=800.0 PL=0
MOVL C00582 V=800.0 PL=0
MOVL C00583 V=800.0 PL=0
MOVL C00584 V=800.0 PL=0
MOVL C00585 V=800.0 PL=0
MOVL C00586 V=800.0 PL=0
MOVL C00587 V=800.0 PL=0
MOVL C00588 V=800.0 PL=0
MOVL C00589 V=800.0 PL=0
MOVL C00590 V=800.0 PL=0
MOVL C00591 V=800.0 PL=0
MOVL C00592 V=800.0 PL=0
MOVL C00593 V=800.0 PL=0
MOVL C00594 V=800.0 PL=0
MOVL C00595 V=800.0 PL=0
MOVL C00596 V=800.0 PL=0
MOVL C00597 V=800.0 PL=0
MOVL C00598 V=800.0 PL=0
MOVL C00599 V=800.0 PL=0
MOVL C00600 V=800.0 PL=0
MOVL C00601 V=800.0 PL=0
MOVL C00602 V=800.0 PL=0
MOVL C00603 V=800.0 PL=0
MOVL C00604 V=800.0 PL=0
MOVL C00605 V=800.0 PL=0
MOVL C00606 V=800.0 PL=0
MOVL C00607 V=800.0 PL=0
MOVL C00608 V=800.0 PL=0
MOVL C00609 V=800.0 PL=0
MOVL C00610 V=800.0 PL=0
MOVL C00611 V=800.0 PL=0
MOVL C00612 V=800.0 PL=0
MOVL C00613 V=800.0 PL=0
MOVL C00614 V=800.0 PL=0
MOVL C00615 V=800.0 PL=0
MOVL C00616 V=800.0 PL=0
MOVL C00617 V=800.0 PL=0
MOVL C00618 V=800.0 PL=0
MOVL C00619 V=800.0 PL=0
MOVL C00620 V=800.0 PL=0
MOVL C00621 V=800.0 PL=0
MOVL C00622 V=800.0 PL=0
MOVL C00623 V=800.0 PL=0
MOVL C00624 V=800.0 PL=0
MOVL C00625 V=800.0 PL=0
MOVL C00626 V=800.0 PL=0
MOVL C00627 V=800.0 PL=0
MOVL C00628 V=800.0 PL=0
MOVL C00629 V=800.0 PL=0
MOVL C00630 V=800.0 PL=0
MOVL C00631 V=800.0 PL=0
MOVL C00632 V=800.0 PL=0
MOVL C00633 V=800.0 PL=0
MOVL C00634 V=800.0 PL=0
MOVL C00635 V=800.0 PL=0
MOVL C00636 V=800.0 PL=0
MOVL C00637 V=800.0 PL=0
MOVL C00638 V=800.0 PL=0
MOVL C00639 V=800.0 PL=0
MOVL C00640 V=800.0 PL=0
MOVL C00641 V=800.0 PL=0
MOVL C00642 V=800.0 PL=0
MOVL C00643 V=800.0 PL=0
MOVL C00644 V=800.0 PL=0
MOVL C00645 V=800.0 PL=0
MOVL C00646 V=800.0 PL=0
MOVL C00647 V=800.0 PL=0
MOVL C00648 V=800.0 PL=0
MOVL C00649 V=800.0 PL=0
MOVL C00650 V=800.0 PL=0
MOVL C00651 V=800.0 PL=0
MOVL C00652 V=800.0 PL=0
MOVL C00653 V=800.0 PL=0
MOVL C00654 V=800.0 PL=0
MOVL C00655 V=800.0 PL=0
MOVL C00656 V=800.0 PL=0
MOVL C00657 V=800.0 PL=0
MOVL C00658 V=800.0 PL=0
MOVL C00659 V=800.0 PL=0
MOVL C00660 V=800.0 PL=0
MOVL C00661 V=800.0 PL=0
MOVL C00662 V=800.0 PL=0
MOVL C00663 V=800.0 PL=0
MOVL C00664 V=800.0 PL=0
MOVL C00665 V=800.0 PL=0
MOVL C00666 V=800.0 PL=0
MOVL C00667 V=800.0 PL=0
MOVL C00668 V=800.0 PL=0
MOVL C00669 V=800.0 PL=0
MOVL C00670 V=800.0 PL=0
MOVL C00671 V=800.0 PL=0
MOVL C00672 V=800.0 PL=0
MOVL C00673 V=800.0 PL=0
MOVL C00674 V=800.0 PL=0
MOVL C00675 V=800.0 PL=0
MOVL C00676 V=800.0 PL=0
MOVL C00677 V=800.0 PL=0
MOVL C00678 V=800.0 PL=0
MOVL C00679 V=800.0 PL=0
MOVL C00680 V=800.0 PL=0
MOVL C00681 V=800.0 PL=0
MOVL C00682 V=800.0 PL=0
MOVL C00683 V=800.0 PL=0
MOVL C00684 V=800.0 PL=0
MOVL C00685 V=800.0 PL=0
MOVL C00686 V=800.0 PL=0
MOVL C00687 V=800.0 PL=0
MOVL C00688 V=800.0 PL=0
MOVL C00689 V=800.0 PL=0
MOVL C00690 V=800.0 PL=0
MOVL C00691 V=800.0 PL=0
MOVL C00692 V=800.0 PL=0
MOVL C00693 V=800.0 PL=0
MOVL C00694 V=800.0 PL=0
MOVL C00695 V=800.0 PL=0
MOVL C00696 V=800.0 PL=0
MOVL C00697 V=800.0 PL=0
MOVL C00698 V=800.0 PL=0
MOVL C00699 V=800.0 PL=0
MOVL C00700 V=800.0 PL=0
MOVL C00701 V=800.0 PL=0
MOVL C00702 V=800.0 PL=0
MOVL C00703 V=800.0 PL=0
MOVL C00704 V=800.0 PL=0
MOVL C00705 V=800.0 PL=0
MOVL C00706 V=800.0 PL=0
MOVL C00707 V=800.0 PL=0
MOVL C00708 V=800.0 PL=0
MOVL C00709 V=800.0 PL=0
MOVL C00710 V=800.0 PL=0
MOVL C00711 V=800.0 PL=0
MOVL C00712 V=800.0 PL=0
MOVL C00713 V=800.0 PL=0
MOVL C00714 V=800.0 PL=0
MOVL C00715 V=800.0 PL=0
MOVL C00716 V=800.0 PL=0
MOVL C00717 V=800.0 PL=0
MOVL C00718 V=800.0 PL=0
MOVL C00719 V=800.0 PL=0
MOVL C00720 V=800.0 PL=0
MOVL C00721 V=800.0 PL=0
MOVL C00722 V=800.0 PL=0
MOVL C00723 V=800.0 PL=0
MOVL C00724 V=800.0 PL=0
MOVL C00725 V=800.0 PL=0
MOVL C00726 V=800.0 PL=0
MOVL C00727 V=800.0 PL=0
MOVL C00728 V=800.0 PL=0
MOVL C00729 V=800.0 PL=0
MOVL C00730 V=800.0 PL=0
MOVL C00731 V=800.0 PL=0
MOVL C00732 V=800.0 PL=0
MOVL C00733 V=800.0 PL=0
MOVL C00734 V=800.0 PL=0
MOVL C00735 V=800.0 PL=0
MOVL C00736 V=800.0 PL=0
MOVL C00737 V=800.0 PL=0
MOVL C00738 V=800.0 PL=0
MOVL C00739 V=800.0 PL=0
MOVL C00740 V=800.0 PL=0
MOVL C00741 V=800.0 PL=0
MOVL C00742 V=800.0 PL=0
MOVL C00743 V=800.0 PL=0
MOVL C00744 V=800.0 PL=0
MOVL C00745 V=800.0 PL=0
MOVL C00746 V=800.0 PL=0
MOVL C00747 V=800.0 PL=0
MOVL C00748 V=800.0 PL=0
MOVL C00749 V=800.0 PL=0
MOVL C00750 V=800.0 PL=0
MOVL C00751 V=800.0 PL=0
MOVL C00752 V=800.0 PL=0
MOVL C00753 V=800.0 PL=0
MOVL C00754 V=800.0 PL=0
MOVL C00755 V=800.0 PL=0
MOVL C00756 V=800.0 PL=0
MOVL C00757 V=800.0 PL=0
MOVL C00758 V=800.0 PL=0
MOVL C00759 V=800.0 PL=0
MOVL C00760 V=800.0 PL=0
MOVL C00761 V=800.0 PL=0
MOVL C00762 V=800.0 PL=0
MOVL C00763 V=800.0 PL=0
MOVL C00764 V=800.0 PL=0
MOVL C00765 V=800.0 PL=0
MOVL C00766 V=800.0 PL=0
MOVL C00767 V=800.0 PL=0
MOVL C00768 V=800.0 PL=0
MOVL C00769 V=800.0 PL=0
MOVL C00770 V=800.0 PL=0
MOVL C00771 V=800.0 PL=0
MOVL C00772 V=800.0 PL=0
MOVL C00773 V=800.0 PL=0
MOVL C00774 V=800.0 PL=0
MOVL C00775 V=800.0 PL=0
MOVL C00776 V=800.0 PL=0
MOVL C00777 V=800.0 PL=0
MOVL C00778 V=800.0 PL=0
MOVL C00779 V=800.0 PL=0
MOVL C00780 V=800.0 PL=0
MOVL C00781 V=800.0 PL=0
MOVL C00782 V=800.0 PL=0
MOVL C00783 V=800.0 PL=0
MOVL C00784 V=800.0 PL=0
MOVL C00785 V=800.0 PL=0
MOVL C00786 V=800.0 PL=0
MOVL C00787 V=800.0 PL=0
MOVL C00788 V=800.0 PL=0
MOVL C00789 V=800.0 PL=0
MOVL C00790 V=800.0 PL=0
MOVL C00791 V=800.0 PL=0
MOVL C00792 V=800.0 PL=0
MOVL C00793 V=800.0 PL=0
MOVL C00794 V=800.0 PL=0
MOVL C00795 V=800.0 PL=0
MOVL C00796 V=800.0 PL=0
MOVL C00797 V=800.0 PL=0
MOVL C00798 V=800.0 PL=0
MOVL C00799 V=800.0 PL=0
MOVL C00800 V=800.0 PL=0
MOVL C00801 V=800.0 PL=0
MOVL C00802 V=800.0 PL=0
MOVL C00803 V=800.0 PL=0
MOVL C00804 V=800.0 PL=0
MOVL C00805 V=800.0 PL=0
MOVL C00806 V=800.0 PL=0
MOVL C00807 V=800.0 PL=0
MOVL C00808 V=800.0 PL=0
MOVL C00809 V=800.0 PL=0
MOVL C00810 V=800.0 PL=0
MOVL C00811 V=800.0 PL=0
MOVL C00812 V=800.0 PL=0
MOVL C00813 V=800.0 PL=0
MOVL C00814 V=800.0 PL=0
MOVL C00815 V=800.0 PL=0
MOVL C00816 V=800.0 PL=0
MOVL C00817 V=800.0 PL=0
MOVL C00818 V=800.0 PL=0
MOVL C00819 V=800.0 PL=0
MOVL C00820 V=800.0 PL=0
MOVL C00821 V=800.0 PL=0
MOVL C00822 V=800.0 PL=0
MOVL C00823 V=800.0 PL=0
MOVL C00824 V=800.0 PL=0
MOVL C00825 V=800.0 PL=0
MOVL C00826 V=800.0 PL=0
MOVL C00827 V=800.0 PL=0
MOVL C00828 V=800.0 PL=0
MOVL C00829 V=800.0 PL=0
MOVL C00830 V=800.0 PL=0
MOVL C00831 V=800.0 PL=0
MOVL C00832 V=800.0 PL=0
MOVL C00833 V=800.0 PL=0
MOVL C00834 V=800.0 PL=0
MOVL C00835 V=800.0 PL=0
MOVL C00836 V=800.0 PL=0
MOVL C00837 V=800.0 PL=0
MOVL C00838 V=800.0 PL=0
MOVL C00839 V=800.0 PL=0
MOVL C00840 V=800.0 PL=0
MOVL C00841 V=800.0 PL=0
MOVL C00842 V=800.0 PL=0
MOVL C00843 V=800.0 PL=0
MOVL C00844 V=800.0 PL=0
MOVL C00845 V=800.0 PL=0
MOVL C00846 V=800.0 PL=0
MOVL C00847 V=800.0 PL=0
MOVL C00848 V=800.0 PL=0
MOVL C00849 V=800.0 PL=0
MOVL C00850 V=800.0 PL=0
MOVL C00851 V=800.0 PL=0
MOVL C00852 V=800.0 PL=0
MOVL C00853 V=800.0 PL=0
MOVL C00854 V=800.0 PL=0
MOVL C00855 V=800.0 PL=0
MOVL C00856 V=800.0 PL=0
MOVL C00857 V=800.0 PL=0
MOVL C00858 V=800.0 PL=0
MOVL C00859 V=800.0 PL=0
MOVL C00860 V=800.0 PL=0
MOVL C00861 V=800.0 PL=0
MOVL C00862 V=800.0 PL=0
MOVL C00863 V=800.0 PL=0
MOVL C00864 V=800.0 PL=0
MOVL C00865 V=800.0 PL=0
MOVL C00866 V=800.0 PL=0
MOVL C00867 V=800.0 PL=0
MOVL C00868 V=800.0 PL=0
MOVL C00869 V=800.0 PL=0
MOVL C00870 V=800.0 PL=0
MOVL C00871 V=800.0 PL=0
MOVL C00872 V=800.0 PL=0
MOVL C00873 V=800.0 PL=0
MOVL C00874 V=800.0 PL=0
MOVL C00875 V=800.0 PL=0
MOVL C00876 V=800.0 PL=0
MOVL C00877 V=800.0 PL=0
MOVL C00878 V=800.0 PL=0
MOVL C00879 V=800.0 PL=0
MOVL C00880 V=800.0 PL=0
MOVL C00881 V=800.0 PL=0
MOVL C00882 V=800.0 PL=0
MOVL C00883 V=800.0 PL=0
MOVL C00884 V=800.0 PL=0
MOVL C00885 V=800.0 PL=0
MOVL C00886 V=800.0 PL=0
MOVL C00887 V=800.0 PL=0
MOVL C00888 V=800.0 PL=0
MOVL C00889 V=800.0 PL=0
MOVL C00890 V=800.0 PL=0
MOVL C00891 V=800.0 PL=0
MOVL C00892 V=800.0 PL=0
MOVL C00893 V=800.0 PL=0
MOVL C00894 V=800.0 PL=0
MOVL C00895 V=800.0 PL=0
MOVL C00896 V=800.0 PL=0
MOVL C00897 V=800.0 PL=0
MOVL C00898 V=800.0 PL=0
MOVL C00899 V=800.0 PL=0
MOVL C00900 V=800.0 PL=0
MOVL C00901 V=800.0 PL=0
MOVL C00902 V=800.0 PL=0
MOVL C00903 V=800.0 PL=0
MOVL C00904 V=800.0 PL=0
MOVL C00905 V=800.0 PL=0
MOVL C00906 V=800.0 PL=0
MOVL C00907 V=800.0 PL=0
MOVL C00908 V=800.0 PL=0
MOVL C00909 V=800.0 PL=0
MOVL C00910 V=800.0 PL=0
MOVL C00911 V=800.0 PL=0
MOVL C00912 V=800.0 PL=0
MOVL C00913 V=800.0 PL=0
MOVL C00914 V=800.0 PL=0
MOVL C00915 V=800.0 PL=0
MOVL C00916 V=800.0 PL=0
MOVL C00917 V=800.0 PL=0
MOVL C00918 V=800.0 PL=0
MOVL C00919 V=800.0 PL=0
MOVL C00920 V=800.0 PL=0
MOVL C00921 V=800.0 PL=0
MOVL C00922 V=800.0 PL=0
MOVL C00923 V=800.0 PL=0
MOVL C00924 V=800.0 PL=0
MOVL C00925 V=800.0 PL=0
MOVL C00926 V=800.0 PL=0
MOVL C00927 V=800.0 PL=0
MOVL C00928 V=800.0 PL=0
MOVL C00929 V=800.0 PL=0
MOVL C00930 V=800.0 PL=0
MOVL C00931 V=800.0 PL=0
MOVL C00932 V=800.0 PL=0
MOVL C00933 V=800.0 PL=0
MOVL C00934 V=800.0 PL=0
MOVL C00935 V=800.0 PL=0
MOVL C00936 V=800.0 PL=0
MOVL C00937 V=800.0 PL=0
MOVL C00938 V=800.0 PL=0
MOVL C00939 V=800.0 PL=0
MOVL C00940 V=800.0 PL=0
MOVL C00941 V=800.0 PL=0
MOVL C00942 V=800.0 PL=0
MOVL C00943 V=800.0 PL=0
MOVL C00944 V=800.0 PL=0
MOVL C00945 V=800.0 PL=0
MOVL C00946 V=800.0 PL=0
MOVL C00947 V=800.0 PL=0
MOVL C00948 V=800.0 PL=0
MOVL C00949 V=800.0 PL=0
MOVL C00950 V=800.0 PL=0
MOVL C00951 V=800.0 PL=0
MOVL C00952 V=800.0 PL=0
MOVL C00953 V=800.0 PL=0
MOVL C00954 V=800.0 PL=0
MOVL C00955 V=800.0 PL=0
MOVL C00956 V=800.0 PL=0
MOVL C00957 V=800.0 PL=0
MOVL C00958 V=800.0 PL=0
MOVL C00959 V=800.0 PL=0
MOVL C00960 V=800.0 PL=0
MOVL C00961 V=800.0 PL=0
MOVL C00962 V=800.0 PL=0
MOVL C00963 V=800.0 PL=0
MOVL C00964 V=800.0 PL=0
MOVL C00965 V=800.0 PL=0
MOVL C00966 V=800.0 PL=0
MOVL C00967 V=800.0 PL=0
MOVL C00968 V=800.0 PL=0
MOVL C00969 V=800.0 PL=0
MOVL C00970 V=800.0 PL=0
MOVL C00971 V=800.0 PL=0
MOVL C00972 V=800.0 PL=0
MOVL C00973 V=800.0 PL=0
MOVL C00974 V=800.0 PL=0
MOVL C00975 V=800.0 PL=0
MOVL C00976 V=800.0 PL=0
MOVL C00977 V=800.0 PL=0
MOVL C00978 V=800.0 PL=0
MOVL C00979 V=800.0 PL=0
MOVL C00980 V=800.0 PL=0
MOVL C00981 V=800.0 PL=0
MOVL C00982 V=800.0 PL=0
MOVL C00983 V=800.0 PL=0
MOVL C00984 V=800.0 PL=0
MOVL C00985 V=800.0 PL=0
MOVL C00986 V=800.0 PL=0
MOVL C00987 V=800.0 PL=0
MOVL C00988 V=800.0 PL=0
MOVL C00989 V=800.0 PL=0
MOVL C00990 V=800.0 PL=0
MOVL C00991 V=800.0 PL=0
MOVL C00992 V=800.0 PL=0
MOVL C00993 V=800.0 PL=0
MOVL C00994 V=800.0 PL=0
MOVL C00995 V=800.0 PL=0
MOVL C00996 V=800.0 PL=0
MOVL C00997 V=800.0 PL=0
MOVL C00998 V=800.0 PL=0
MOVL C00999 V=800.0 PL=0
MOVL C01000 V=800.0 PL=0
MOVL C01001 V=800.0 PL=0
MOVL C01002 V=800.0 PL=0
MOVL C01003 V=800.0 PL=0
MOVL C01004 V=800.0 PL=0
MOVL C01005 V=800.0 PL=0
MOVL C01006 V=800.0 PL=0
MOVL C01007 V=800.0 PL=0
MOVL C01008 V=800.0 PL=0
MOVL C01009 V=800.0 PL=0
MOVL C01010 V=800.0 PL=0
MOVL C01011 V=800.0 PL=0
MOVL C01012 V=800.0 PL=0
MOVL C01013 V=800.0 PL=0
MOVL C01014 V=800.0 PL=0
MOVL C01015 V=800.0 PL=0
MOVL C01016 V=800.0 PL=0
MOVL C01017 V=800.0 PL=0
MOVL C01018 V=800.0 PL=0
MOVL C01019 V=800.0 PL=0
MOVL C01020 V=800.0 PL=0
MOVL C01021 V=800.0 PL=0
MOVL C01022 V=800.0 PL=0
MOVL C01023 V=800.0 PL=0
MOVL C01024 V=800.0 PL=0
MOVL C01025 V=800.0 PL=0
MOVL C01026 V=800.0 PL=0
MOVL C01027 V=800.0 PL=0
MOVL C01028 V=800.0 PL=0
MOVL C01029 V=800.0 PL=0
MOVL C01030 V=800.0 PL=0
MOVL C01031 V=800.0 PL=0
MOVL C01032 V=800.0 PL=0
MOVL C01033 V=800.0 PL=0
MOVL C01034 V=800.0 PL=0
MOVL C01035 V=800.0 PL=0
MOVL C01036 V=800.0 PL=0
MOVL C01037 V=800.0 PL=0
MOVL C01038 V=800.0 PL=0
MOVL C01039 V=800.0 PL=0
MOVL C01040 V=800.0 PL=0
MOVL C01041 V=800.0 PL=0
MOVL C01042 V=800.0 PL=0
MOVL C01043 V=800.0 PL=0
MOVL C01044 V=800.0 PL=0
MOVL C01045 V=800.0 PL=0
MOVL C01046 V=800.0 PL=0
MOVL C01047 V=800.0 PL=0
MOVL C01048 V=800.0 PL=0
MOVL C01049 V=800.0 PL=0
MOVL C01050 V=800.0 PL=0
MOVL C01051 V=800.0 PL=0
MOVL C01052 V=800.0 PL=0
MOVL C01053 V=800.0 PL=0
MOVL C01054 V=800.0 PL=0
MOVL C01055 V=800.0 PL=0
MOVL C01056 V=800.0 PL=0
MOVL C01057 V=800.0 PL=0
MOVL C01058 V=800.0 PL=0
MOVL C01059 V=800.0 PL=0
MOVL C01060 V=800.0 PL=0
MOVL C01061 V=800.0 PL=0
MOVL C01062 V=800.0 PL=0
MOVL C01063 V=800.0 PL=0
MOVL C01064 V=800.0 PL=0
MOVL C01065 V=800.0 PL=0
MOVL C01066 V=800.0 PL=0
MOVL C01067 V=800.0 PL=0
MOVL C01068 V=800.0 PL=0
MOVL C01069 V=800.0 PL=0
MOVL C01070 V=800.0 PL=0
MOVL C01071 V=800.0 PL=0
MOVL C01072 V=800.0 PL=0
MOVL C01073 V=800.0 PL=0
MOVL C01074 V=800.0 PL=0
MOVL C01075 V=800.0 PL=0
MOVL C01076 V=800.0 PL=0
MOVL C01077 V=800.0 PL=0
MOVL C01078 V=800.0 PL=0
MOVL C01079 V=800.0 PL=0
MOVL C01080 V=800.0 PL=0
MOVL C01081 V=800.0 PL=0
MOVL C01082 V=800.0 PL=0
MOVL C01083 V=800.0 PL=0
MOVL C01084 V=800.0 PL=0
MOVL C01085 V=800.0 PL=0
MOVL C01086 V=800.0 PL=0
MOVL C01087 V=800.0 PL=0
MOVL C01088 V=800.0 PL=0
MOVL C01089 V=800.0 PL=0
MOVL C01090 V=800.0 PL=0
MOVL C01091 V=800.0 PL=0
MOVL C01092 V=800.0 PL=0
MOVL C01093 V=800.0 PL=0
MOVL C01094 V=800.0 PL=0
MOVL C01095 V=800.0 PL=0
MOVL C01096 V=800.0 PL=0
MOVL C01097 V=800.0 PL=0
MOVL C01098 V=800.0 PL=0
MOVL C01099 V=800.0 PL=0
MOVL C01100 V=800.0 PL=0
MOVL C01101 V=800.0 PL=0
MOVL C01102 V=800.0 PL=0
MOVL C01103 V=800.0 PL=0
MOVL C01104 V=800.0 PL=0
MOVL C01105 V=800.0 PL=0
MOVL C01106 V=800.0 PL=0
MOVL C01107 V=800.0 PL=0
MOVL C01108 V=800.0 PL=0
MOVL C01109 V=800.0 PL=0
MOVL C01110 V=800.0 PL=0
MOVL C01111 V=800.0 PL=0
MOVL C01112 V=800.0 PL=0
MOVL C01113 V=800.0 PL=0
MOVL C01114 V=800.0 PL=0
MOVL C01115 V=800.0 PL=0
MOVL C01116 V=800.0 PL=0
MOVL C01117 V=800.0 PL=0
MOVL C01118 V=800.0 PL=0
MOVL C01119 V=800.0 PL=0
MOVL C01120 V=800.0 PL=0
MOVL C01121 V=800.0 PL=0
MOVL C01122 V=800.0 PL=0
MOVL C01123 V=800.0 PL=0
MOVL C01124 V=800.0 PL=0
MOVL C01125 V=800.0 PL=0
MOVL C01126 V=800.0 PL=0
MOVL C01127 V=800.0 PL=0
MOVL C01128 V=800.0 PL=0
MOVL C01129 V=800.0 PL=0
MOVL C01130 V=800.0 PL=0
MOVL C01131 V=800.0 PL=0
MOVL C01132 V=800.0 PL=0
MOVL C01133 V=800.0 PL=0
MOVL C01134 V=800.0 PL=0
MOVL C01135 V=800.0 PL=0
MOVL C01136 V=800.0 PL=0
MOVL C01137 V=800.0 PL=0
MOVL C01138 V=800.0 PL=0
MOVL C01139 V=800.0 PL=0
MOVL C01140 V=800.0 PL=0
MOVL C01141 V=800.0 PL=0
MOVL C01142 V=800.0 PL=0
MOVL C01143 V=800.0 PL=0
MOVL C01144 V=800.0 PL=0
MOVL C01145 V=800.0 PL=0
MOVL C01146 V=800.0 PL=0
MOVL C01147 V=800.0 PL=0
MOVL C01148 V=800.0 PL=0
MOVL C01149 V=800.0 PL=0
MOVL C01150 V=800.0 PL=0
MOVL C01151 V=800.0 PL=0
MOVL C01152 V=800.0 PL=0
MOVL C01153 V=800.0 PL=0
MOVL C01154 V=800.0 PL=0
MOVL C01155 V=800.0 PL=0
MOVL C01156 V=800.0 PL=0
MOVL C01157 V=800.0 PL=0
MOVL C01158 V=800.0 PL=0
MOVL C01159 V=800.0 PL=0
MOVL C01160 V=800.0 PL=0
MOVL C01161 V=800.0 PL=0
MOVL C01162 V=800.0 PL=0
MOVL C01163 V=800.0 PL=0
MOVL C01164 V=800.0 PL=0
MOVL C01165 V=800.0 PL=0
MOVL C01166 V=800.0 PL=0
MOVL C01167 V=800.0 PL=0
MOVL C01168 V=800.0 PL=0
MOVL C01169 V=800.0 PL=0
MOVL C01170 V=800.0 PL=0
MOVL C01171 V=800.0 PL=0
MOVL C01172 V=800.0 PL=0
MOVL C01173 V=800.0 PL=0
MOVL C01174 V=800.0 PL=0
MOVL C01175 V=800.0 PL=0
MOVL C01176 V=800.0 PL=0
MOVL C01177 V=800.0 PL=0
MOVL C01178 V=800.0 PL=0
MOVL C01179 V=800.0 PL=0
MOVL C01180 V=800.0 PL=0
MOVL C01181 V=800.0 PL=0
MOVL C01182 V=800.0 PL=0
MOVL C01183 V=800.0 PL=0
MOVL C01184 V=800.0 PL=0
MOVL C01185 V=800.0 PL=0
MOVL C01186 V=800.0 PL=0
MOVL C01187 V=800.0 PL=0
MOVL C01188 V=800.0 PL=0
MOVL C01189 V=800.0 PL=0
MOVL C01190 V=800.0 PL=0
MOVL C01191 V=800.0 PL=0
MOVL C01192 V=800.0 PL=0
MOVL C01193 V=800.0 PL=0
MOVL C01194 V=800.0 PL=0
MOVL C01195 V=800.0 PL=0
MOVL C01196 V=800.0 PL=0
MOVL C01197 V=800.0 PL=0
MOVL C01198 V=800.0 PL=0
MOVL C01199 V=800.0 PL=0
MOVL C01200 V=800.0 PL=0
MOVL C01201 V=800.0 PL=0
MOVL C01202 V=800.0 PL=0
MOVL C01203 V=800.0 PL=0
MOVL C01204 V=800.0 PL=0
MOVL C01205 V=800.0 PL=0
MOVL C01206 V=800.0 PL=0
MOVL C01207 V=800.0 PL=0
MOVL C01208 V=800.0 PL=0
MOVL C01209 V=800.0 PL=0
MOVL C01210 V=800.0 PL=0
MOVL C01211 V=800.0 PL=0
MOVL C01212 V=800.0 PL=0
MOVL C01213 V=800.0 PL=0
MOVL C01214 V=800.0 PL=0
MOVL C01215 V=800.0 PL=0
MOVL C01216 V=800.0 PL=0
MOVL C01217 V=800.0 PL=0
MOVL C01218 V=800.0 PL=0
MOVL C01219 V=800.0 PL=0
MOVL C01220 V=800.0 PL=0
MOVL C01221 V=800.0 PL=0
MOVL C01222 V=800.0 PL=0
MOVL C01223 V=800.0 PL=0
MOVL C01224 V=800.0 PL=0
MOVL C01225 V=800.0 PL=0
MOVL C01226 V=800.0 PL=0
MOVL C01227 V=800.0 PL=0
MOVL C01228 V=800.0 PL=0
MOVL C01229 V=800.0 PL=0
MOVL C01230 V=800.0 PL=0
MOVL C01231 V=800.0 PL=0
MOVL C01232 V=800.0 PL=0
MOVL C01233 V=800.0 PL=0
MOVL C01234 V=800.0 PL=0
MOVL C01235 V=800.0 PL=0
MOVL C01236 V=800.0 PL=0
MOVL C01237 V=800.0 PL=0
MOVL C01238 V=800.0 PL=0
MOVL C01239 V=800.0 PL=0
MOVL C01240 V=800.0 PL=0
MOVL C01241 V=800.0 PL=0
MOVL C01242 V=800.0 PL=0
MOVL C01243 V=800.0 PL=0
MOVL C01244 V=800.0 PL=0
MOVL C01245 V=800.0 PL=0
MOVL C01246 V=800.0 PL=0
MOVL C01247 V=800.0 PL=0
MOVL C01248 V=800.0 PL=0
MOVL C01249 V=800.0 PL=0
MOVL C01250 V=800.0 PL=0
MOVL C01251 V=800.0 PL=0
MOVL C01252 V=800.0 PL=0
MOVL C01253 V=800.0 PL=0
MOVL C01254 V=800.0 PL=0
MOVL C01255 V=800.0 PL=0
MOVL C01256 V=800.0 PL=0
MOVL C01257 V=800.0 PL=0
MOVL C01258 V=800.0 PL=0
MOVL C01259 V=800.0 PL=0
MOVL C01260 V=800.0 PL=0
MOVL C01261 V=800.0 PL=0
MOVL C01262 V=800.0 PL=0
MOVL C01263 V=800.0 PL=0
MOVL C01264 V=800.0 PL=0
MOVL C01265 V=800.0 PL=0
MOVL C01266 V=800.0 PL=0
MOVL C01267 V=800.0 PL=0
MOVL C01268 V=800.0 PL=0
MOVL C01269 V=800.0 PL=0
MOVL C01270 V=800.0 PL=0
MOVL C01271 V=800.0 PL=0
MOVL C01272 V=800.0 PL=0
MOVL C01273 V=800.0 PL=0
MOVL C01274 V=800.0 PL=0
MOVL C01275 V=800.0 PL=0
MOVL C01276 V=800.0 PL=0
MOVL C01277 V=800.0 PL=0
MOVL C01278 V=800.0 PL=0
MOVL C01279 V=800.0 PL=0
MOVL C01280 V=800.0 PL=0
MOVL C01281 V=800.0 PL=0
MOVL C01282 V=800.0 PL=0
MOVL C01283 V=800.0 PL=0
MOVL C01284 V=800.0 PL=0
MOVL C01285 V=800.0 PL=0
MOVL C01286 V=800.0 PL=0
MOVL C01287 V=800.0 PL=0
MOVL C01288 V=800.0 PL=0
MOVL C01289 V=800.0 PL=0
MOVL C01290 V=800.0 PL=0
MOVL C01291 V=800.0 PL=0
MOVL C01292 V=800.0 PL=0
MOVL C01293 V=800.0 PL=0
MOVL C01294 V=800.0 PL=0
MOVL C01295 V=800.0 PL=0
MOVL C01296 V=800.0 PL=0
MOVL C01297 V=800.0 PL=0
MOVL C01298 V=800.0 PL=0
MOVL C01299 V=800.0 PL=0
MOVL C01300 V=800.0 PL=0
MOVL C01301 V=800.0 PL=0
MOVL C01302 V=800.0 PL=0
MOVL C01303 V=800.0 PL=0
MOVL C01304 V=800.0 PL=0
MOVL C01305 V=800.0 PL=0
MOVL C01306 V=800.0 PL=0
MOVL C01307 V=800.0 PL=0
MOVL C01308 V=800.0 PL=0
MOVL C01309 V=800.0 PL=0
MOVL C01310 V=800.0 PL=0
MOVL C01311 V=800.0 PL=0
MOVL C01312 V=800.0 PL=0
MOVL C01313 V=800.0 PL=0
MOVL C01314 V=800.0 PL=0
MOVL C01315 V=800.0 PL=0
MOVL C01316 V=800.0 PL=0
MOVL C01317 V=800.0 PL=0
MOVL C01318 V=800.0 PL=0
MOVL C01319 V=800.0 PL=0
MOVL C01320 V=800.0 PL=0
MOVL C01321 V=800.0 PL=0
MOVL C01322 V=800.0 PL=0
MOVL C01323 V=800.0 PL=0
MOVL C01324 V=800.0 PL=0
MOVL C01325 V=800.0 PL=0
MOVL C01326 V=800.0 PL=0
MOVL C01327 V=800.0 PL=0
MOVL C01328 V=800.0 PL=0
MOVL C01329 V=800.0 PL=0
MOVL C01330 V=800.0 PL=0
MOVL C01331 V=800.0 PL=0
MOVL C01332 V=800.0 PL=0
MOVL C01333 V=800.0 PL=0
MOVL C01334 V=800.0 PL=0
MOVL C01335 V=800.0 PL=0
MOVL C01336 V=800.0 PL=0
MOVL C01337 V=800.0 PL=0
MOVL C01338 V=800.0 PL=0
MOVL C01339 V=800.0 PL=0
MOVL C01340 V=800.0 PL=0
MOVL C01341 V=800.0 PL=0
MOVL C01342 V=800.0 PL=0
MOVL C01343 V=800.0 PL=0
MOVL C01344 V=800.0 PL=0
MOVL C01345 V=800.0 PL=0
MOVL C01346 V=800.0 PL=0
MOVL C01347 V=800.0 PL=0
MOVL C01348 V=800.0 PL=0
MOVL C01349 V=800.0 PL=0
MOVL C01350 V=800.0 PL=0
MOVL C01351 V=800.0 PL=0
MOVL C01352 V=800.0 PL=0
MOVL C01353 V=800.0 PL=0
MOVL C01354 V=800.0 PL=0
MOVL C01355 V=800.0 PL=0
MOVL C01356 V=800.0 PL=0
MOVL C01357 V=800.0 PL=0
MOVL C01358 V=800.0 PL=0
MOVL C01359 V=800.0 PL=0
MOVL C01360 V=800.0 PL=0
MOVL C01361 V=800.0 PL=0
MOVL C01362 V=800.0 PL=0
MOVL C01363 V=800.0 PL=0
MOVL C01364 V=800.0 PL=0
MOVL C01365 V=800.0 PL=0
MOVL C01366 V=800.0 PL=0
MOVL C01367 V=800.0 PL=0
MOVL C01368 V=800.0 PL=0
MOVL C01369 V=800.0 PL=0
MOVL C01370 V=800.0 PL=0
MOVL C01371 V=800.0 PL=0
MOVL C01372 V=800.0 PL=0
MOVL C01373 V=800.0 PL=0
MOVL C01374 V=800.0 PL=0
MOVL C01375 V=800.0 PL=0
MOVL C01376 V=800.0 PL=0
MOVL C01377 V=800.0 PL=0
MOVL C01378 V=800.0 PL=0
MOVL C01379 V=800.0 PL=0
MOVL C01380 V=800.0 PL=0
MOVL C01381 V=800.0 PL=0
MOVL C01382 V=800.0 PL=0
MOVL C01383 V=800.0 PL=0
MOVL C01384 V=800.0 PL=0
MOVL C01385 V=800.0 PL=0
MOVL C01386 V=800.0 PL=0
MOVL C01387 V=800.0 PL=0
MOVL C01388 V=800.0 PL=0
MOVL C01389 V=800.0 PL=0
MOVL C01390 V=800.0 PL=0
MOVL C01391 V=800.0 PL=0
MOVL C01392 V=800.0 PL=0
MOVL C01393 V=800.0 PL=0
MOVL C01394 V=800.0 PL=0
MOVL C01395 V=800.0 PL=0
MOVL C01396 V=800.0 PL=0
MOVL C01397 V=800.0 PL=0
MOVL C01398 V=800.0 PL=0
MOVL C01399 V=800.0 PL=0
MOVL C01400 V=800.0 PL=0
MOVL C01401 V=800.0 PL=0
MOVL C01402 V=800.0 PL=0
MOVL C01403 V=800.0 PL=0
MOVL C01404 V=800.0 PL=0
MOVL C01405 V=800.0 PL=0
MOVL C01406 V=800.0 PL=0
MOVL C01407 V=800.0 PL=0
MOVL C01408 V=800.0 PL=0
MOVL C01409 V=800.0 PL=0
MOVL C01410 V=800.0 PL=0
MOVL C01411 V=800.0 PL=0
MOVL C01412 V=800.0 PL=0
MOVL C01413 V=800.0 PL=0
MOVL C01414 V=800.0 PL=0
MOVL C01415 V=800.0 PL=0
MOVL C01416 V=800.0 PL=0
MOVL C01417 V=800.0 PL=0
MOVL C01418 V=800.0 PL=0
MOVL C01419 V=800.0 PL=0
MOVL C01420 V=800.0 PL=0
MOVL C01421 V=800.0 PL=0
MOVL C01422 V=800.0 PL=0
MOVL C01423 V=800.0 PL=0
MOVL C01424 V=800.0 PL=0
MOVL C01425 V=800.0 PL=0
MOVL C01426 V=800.0 PL=0
MOVL C01427 V=800.0 PL=0
MOVL C01428 V=800.0 PL=0
MOVL C01429 V=800.0 PL=0
MOVL C01430 V=800.0 PL=0
MOVL C01431 V=800.0 PL=0
MOVL C01432 V=800.0 PL=0
MOVL C01433 V=800.0 PL=0
MOVL C01434 V=800.0 PL=0
MOVL C01435 V=800.0 PL=0
MOVL C01436 V=800.0 PL=0
MOVL C01437 V=800.0 PL=0
MOVL C01438 V=800.0 PL=0
MOVL C01439 V=800.0 PL=0
MOVL C01440 V=800.0 PL=0
MOVL C01441 V=800.0 PL=0
MOVL C01442 V=800.0 PL=0
MOVL C01443 V=800.0 PL=0
MOVL C01444 V=800.0 PL=0
MOVL C01445 V=800.0 PL=0
MOVL C01446 V=800.0 PL=0
MOVL C01447 V=800.0 PL=0
MOVL C01448 V=800.0 PL=0
MOVL C01449 V=800.0 PL=0
MOVL C01450 V=800.0 PL=0
MOVL C01451 V=800.0 PL=0
MOVL C01452 V=800.0 PL=0
MOVL C01453 V=800.0 PL=0
MOVL C01454 V=800.0 PL=0
MOVL C01455 V=800.0 PL=0
MOVL C01456 V=800.0 PL=0
MOVL C01457 V=800.0 PL=0
MOVL C01458 V=800.0 PL=0
MOVL C01459 V=800.0 PL=0
MOVL C01460 V=800.0 PL=0
MOVL C01461 V=800.0 PL=0
MOVL C01462 V=800.0 PL=0
MOVL C01463 V=800.0 PL=0
MOVL C01464 V=800.0 PL=0
MOVL C01465 V=800.0 PL=0
MOVL C01466 V=800.0 PL=0
MOVL C01467 V=800.0 PL=0
MOVL C01468 V=800.0 PL=0
MOVL C01469 V=800.0 PL=0
MOVL C01470 V=800.0 PL=0
MOVL C01471 V=800.0 PL=0
MOVL C01472 V=800.0 PL=0
MOVL C01473 V=800.0 PL=0
MOVL C01474 V=800.0 PL=0
MOVL C01475 V=800.0 PL=0
MOVL C01476 V=800.0 PL=0
MOVL C01477 V=800.0 PL=0
MOVL C01478 V=800.0 PL=0
MOVL C01479 V=800.0 PL=0
MOVL C01480 V=800.0 PL=0
MOVL C01481 V=800.0 PL=0
MOVL C01482 V=800.0 PL=0
MOVL C01483 V=800.0 PL=0
MOVL C01484 V=800.0 PL=0
MOVL C01485 V=800.0 PL=0
MOVL C01486 V=800.0 PL=0
MOVL C01487 V=800.0 PL=0
MOVL C01488 V=800.0 PL=0
MOVL C01489 V=800.0 PL=0
MOVL C01490 V=800.0 PL=0
MOVL C01491 V=800.0 PL=0
MOVL C01492 V=800.0 PL=0
MOVL C01493 V=800.0 PL=0
MOVL C01494 V=800.0 PL=0
MOVL C01495 V=800.0 PL=0
MOVL C01496 V=800.0 PL=0
MOVL C01497 V=800.0 PL=0
MOVL C01498 V=800.0 PL=0
MOVL C01499 V=800.0 PL=0
MOVL C01500 V=800.0 PL=0
MOVL C01501 V=800.0 PL=0
MOVL C01502 V=800.0 PL=0
MOVL C01503 V=800.0 PL=0
MOVL C01504 V=800.0 PL=0
MOVL C01505 V=800.0 PL=0
MOVL C01506 V=800.0 PL=0
MOVL C01507 V=800.0 PL=0
MOVL C01508 V=800.0 PL=0
MOVL C01509 V=800.0 PL=0
MOVL C01510 V=800.0 PL=0
MOVL C01511 V=800.0 PL=0
MOVL C01512 V=800.0 PL=0
MOVL C01513 V=800.0 PL=0
MOVL C01514 V=800.0 PL=0
MOVL C01515 V=800.0 PL=0
MOVL C01516 V=800.0 PL=0
MOVL C01517 V=800.0 PL=0
MOVL C01518 V=800.0 PL=0
MOVL C01519 V=800.0 PL=0
MOVL C01520 V=800.0 PL=0
MOVL C01521 V=800.0 PL=0
MOVL C01522 V=800.0 PL=0
MOVL C01523 V=800.0 PL=0
MOVL C01524 V=800.0 PL=0
MOVL C01525 V=800.0 PL=0
MOVL C01526 V=800.0 PL=0
MOVL C01527 V=800.0 PL=0
MOVL C01528 V=800.0 PL=0
MOVL C01529 V=800.0 PL=0
MOVL C01530 V=800.0 PL=0
MOVL C01531 V=800.0 PL=0
MOVL C01532 V=800.0 PL=0
MOVL C01533 V=800.0 PL=0
MOVL C01534 V=800.0 PL=0
MOVL C01535 V=800.0 PL=0
MOVL C01536 V=800.0 PL=0
MOVL C01537 V=800.0 PL=0
MOVL C01538 V=800.0 PL=0
MOVL C01539 V=800.0 PL=0
MOVL C01540 V=800.0 PL=0
MOVL C01541 V=800.0 PL=0
MOVL C01542 V=800.0 PL=0
MOVL C01543 V=800.0 PL=0
MOVL C01544 V=800.0 PL=0
MOVL C01545 V=800.0 PL=0
MOVL C01546 V=800.0 PL=0
MOVL C01547 V=800.0 PL=0
MOVL C01548 V=800.0 PL=0
MOVL C01549 V=800.0 PL=0
MOVL C01550 V=800.0 PL=0
MOVL C01551 V=800.0 PL=0
MOVL C01552 V=800.0 PL=0
MOVL C01553 V=800.0 PL=0
MOVL C01554 V=800.0 PL=0
MOVL C01555 V=800.0 PL=0
MOVL C01556 V=800.0 PL=0
MOVL C01557 V=800.0 PL=0
MOVL C01558 V=800.0 PL=0
MOVL C01559 V=800.0 PL=0
MOVL C01560 V=800.0 PL=0
MOVL C01561 V=800.0 PL=0
MOVL C01562 V=800.0 PL=0
MOVL C01563 V=800.0 PL=0
MOVL C01564 V=800.0 PL=0
MOVL C01565 V=800.0 PL=0
MOVL C01566 V=800.0 PL=0
MOVL C01567 V=800.0 PL=0
MOVL C01568 V=800.0 PL=0
MOVL C01569 V=800.0 PL=0
MOVL C01570 V=800.0 PL=0
MOVL C01571 V=800.0 PL=0
MOVL C01572 V=800.0 PL=0
MOVL C01573 V=800.0 PL=0
MOVL C01574 V=800.0 PL=0
MOVL C01575 V=800.0 PL=0
MOVL C01576 V=800.0 PL=0
MOVL C01577 V=800.0 PL=0
MOVL C01578 V=800.0 PL=0
MOVL C01579 V=800.0 PL=0
MOVL C01580 V=800.0 PL=0
MOVL C01581 V=800.0 PL=0
MOVL C01582 V=800.0 PL=0
MOVL C01583 V=800.0 PL=0
MOVL C01584 V=800.0 PL=0
MOVL C01585 V=800.0 PL=0
MOVL C01586 V=800.0 PL=0
MOVL C01587 V=800.0 PL=0
MOVL C01588 V=800.0 PL=0
MOVL C01589 V=800.0 PL=0
MOVL C01590 V=800.0 PL=0
MOVL C01591 V=800.0 PL=0
MOVL C01592 V=800.0 PL=0
MOVL C01593 V=800.0 PL=0
MOVL C01594 V=800.0 PL=0
MOVL C01595 V=800.0 PL=0
MOVL C01596 V=800.0 PL=0
MOVL C01597 V=800.0 PL=0
MOVL C01598 V=800.0 PL=0
MOVL C01599 V=800.0 PL=0
MOVL C01600 V=800.0 PL=0
MOVL C01601 V=800.0 PL=0
MOVL C01602 V=800.0 PL=0
MOVL C01603 V=800.0 PL=0
MOVL C01604 V=800.0 PL=0
MOVL C01605 V=800.0 PL=0
MOVL C01606 V=800.0 PL=0
MOVL C01607 V=800.0 PL=0
MOVL C01608 V=800.0 PL=0
MOVL C01609 V=800.0 PL=0
MOVL C01610 V=800.0 PL=0
MOVL C01611 V=800.0 PL=0
MOVL C01612 V=800.0 PL=0
MOVL C01613 V=800.0 PL=0
MOVL C01614 V=800.0 PL=0
MOVL C01615 V=800.0 PL=0
MOVL C01616 V=800.0 PL=0
MOVL C01617 V=800.0 PL=0
MOVL C01618 V=800.0 PL=0
MOVL C01619 V=800.0 PL=0
MOVL C01620 V=800.0 PL=0
MOVL C01621 V=800.0 PL=0
MOVL C01622 V=800.0 PL=0
MOVL C01623 V=800.0 PL=0
MOVL C01624 V=800.0 PL=0
MOVL C01625 V=800.0 PL=0
MOVL C01626 V=800.0 PL=0
MOVL C01627 V=800.0 PL=0
MOVL C01628 V=800.0 PL=0
MOVL C01629 V=800.0 PL=0
MOVL C01630 V=800.0 PL=0
MOVL C01631 V=800.0 PL=0
MOVL C01632 V=800.0 PL=0
MOVL C01633 V=800.0 PL=0
MOVL C01634 V=800.0 PL=0
MOVL C01635 V=800.0 PL=0
MOVL C01636 V=800.0 PL=0
MOVL C01637 V=800.0 PL=0
MOVL C01638 V=800.0 PL=0
MOVL C01639 V=800.0 PL=0
MOVL C01640 V=800.0 PL=0
MOVL C01641 V=800.0 PL=0
MOVL C01642 V=800.0 PL=0
MOVL C01643 V=800.0 PL=0
MOVL C01644 V=800.0 PL=0
MOVL C01645 V=800.0 PL=0
MOVL C01646 V=800.0 PL=0
MOVL C01647 V=800.0 PL=0
MOVL C01648 V=800.0 PL=0
MOVL C01649 V=800.0 PL=0
MOVL C01650 V=800.0 PL=0
MOVL C01651 V=800.0 PL=0
MOVL C01652 V=800.0 PL=0
MOVL C01653 V=800.0 PL=0
MOVL C01654 V=800.0 PL=0
MOVL C01655 V=800.0 PL=0
MOVL C01656 V=800.0 PL=0
MOVL C01657 V=800.0 PL=0
MOVL C01658 V=800.0 PL=0
MOVL C01659 V=800.0 PL=0
MOVL C01660 V=800.0 PL=0
MOVL C01661 V=800.0 PL=0
MOVL C01662 V=800.0 PL=0
MOVL C01663 V=800.0 PL=0
MOVL C01664 V=800.0 PL=0
MOVL C01665 V=800.0 PL=0
MOVL C01666 V=800.0 PL=0
MOVL C01667 V=800.0 PL=0
MOVL C01668 V=800.0 PL=0
MOVL C01669 V=800.0 PL=0
MOVL C01670 V=800.0 PL=0
MOVL C01671 V=800.0 PL=0
MOVL C01672 V=800.0 PL=0
MOVL C01673 V=800.0 PL=0
MOVL C01674 V=800.0 PL=0
MOVL C01675 V=800.0 PL=0
MOVL C01676 V=800.0 PL=0
MOVL C01677 V=800.0 PL=0
MOVL C01678 V=800.0 PL=0
MOVL C01679 V=800.0 PL=0
MOVL C01680 V=800.0 PL=0
MOVL C01681 V=800.0 PL=0
MOVL C01682 V=800.0 PL=0
MOVL C01683 V=800.0 PL=0
MOVL C01684 V=800.0 PL=0
MOVL C01685 V=800.0 PL=0
MOVL C01686 V=800.0 PL=0
MOVL C01687 V=800.0 PL=0
MOVL C01688 V=800.0 PL=0
MOVL C01689 V=800.0 PL=0
MOVL C01690 V=800.0 PL=0
MOVL C01691 V=800.0 PL=0
MOVL C01692 V=800.0 PL=0
MOVL C01693 V=800.0 PL=0
MOVL C01694 V=800.0 PL=0
MOVL C01695 V=800.0 PL=0
MOVL C01696 V=800.0 PL=0
MOVL C01697 V=800.0 PL=0
MOVL C01698 V=800.0 PL=0
MOVL C01699 V=800.0 PL=0
MOVL C01700 V=800.0 PL=0
MOVL C01701 V=800.0 PL=0
MOVL C01702 V=800.0 PL=0
MOVL C01703 V=800.0 PL=0
MOVL C01704 V=800.0 PL=0
MOVL C01705 V=800.0 PL=0
MOVL C01706 V=800.0 PL=0
MOVL C01707 V=800.0 PL=0
MOVL C01708 V=800.0 PL=0
MOVL C01709 V=800.0 PL=0
MOVL C01710 V=800.0 PL=0
MOVL C01711 V=800.0 PL=0
MOVL C01712 V=800.0 PL=0
MOVL C01713 V=800.0 PL=0
MOVL C01714 V=800.0 PL=0
MOVL C01715 V=800.0 PL=0
MOVL C01716 V=800.0 PL=0
MOVL C01717 V=800.0 PL=0
MOVL C01718 V=800.0 PL=0
MOVL C01719 V=800.0 PL=0
MOVL C01720 V=800.0 PL=0
MOVL C01721 V=800.0 PL=0
MOVL C01722 V=800.0 PL=0
MOVL C01723 V=800.0 PL=0
MOVL C01724 V=800.0 PL=0
MOVL C01725 V=800.0 PL=0
MOVL C01726 V=800.0 PL=0
MOVL C01727 V=800.0 PL=0
MOVL C01728 V=800.0 PL=0
MOVL C01729 V=800.0 PL=0
MOVL C01730 V=800.0 PL=0
MOVL C01731 V=800.0 PL=0
MOVL C01732 V=800.0 PL=0
MOVL C01733 V=800.0 PL=0
MOVL C01734 V=800.0 PL=0
MOVL C01735 V=800.0 PL=0
MOVL C01736 V=800.0 PL=0
MOVL C01737 V=800.0 PL=0
MOVL C01738 V=800.0 PL=0
MOVL C01739 V=800.0 PL=0
MOVL C01740 V=800.0 PL=0
MOVL C01741 V=800.0 PL=0
MOVL C01742 V=800.0 PL=0
MOVL C01743 V=800.0 PL=0
MOVL C01744 V=800.0 PL=0
MOVL C01745 V=800.0 PL=0
MOVL C01746 V=800.0 PL=0
MOVL C01747 V=800.0 PL=0
MOVL C01748 V=800.0 PL=0
MOVL C01749 V=800.0 PL=0
MOVL C01750 V=800.0 PL=0
MOVL C01751 V=800.0 PL=0
MOVL C01752 V=800.0 PL=0
MOVL C01753 V=800.0 PL=0
MOVL C01754 V=800.0 PL=0
MOVL C01755 V=800.0 PL=0
MOVL C01756 V=800.0 PL=0
MOVL C01757 V=800.0 PL=0
MOVL C01758 V=800.0 PL=0
MOVL C01759 V=800.0 PL=0
MOVL C01760 V=800.0 PL=0
MOVL C01761 V=800.0 PL=0
MOVL C01762 V=800.0 PL=0
MOVL C01763 V=800.0 PL=0
MOVL C01764 V=800.0 PL=0
MOVL C01765 V=800.0 PL=0
MOVL C01766 V=800.0 PL=0
MOVL C01767 V=800.0 PL=0
MOVL C01768 V=800.0 PL=0
MOVL C01769 V=800.0 PL=0
MOVL C01770 V=800.0 PL=0
MOVL C01771 V=800.0 PL=0
MOVL C01772 V=800.0 PL=0
MOVL C01773 V=800.0 PL=0
MOVL C01774 V=800.0 PL=0
MOVL C01775 V=800.0 PL=0
MOVL C01776 V=800.0 PL=0
MOVL C01777 V=800.0 PL=0
MOVL C01778 V=800.0 PL=0
MOVL C01779 V=800.0 PL=0
MOVL C01780 V=800.0 PL=0
MOVL C01781 V=800.0 PL=0
MOVL C01782 V=800.0 PL=0
MOVL C01783 V=800.0 PL=0
MOVL C01784 V=800.0 PL=0
MOVL C01785 V=800.0 PL=0
MOVL C01786 V=800.0 PL=0
MOVL C01787 V=800.0 PL=0
MOVL C01788 V=800.0 PL=0
MOVL C01789 V=800.0 PL=0
MOVL C01790 V=800.0 PL=0
MOVL C01791 V=800.0 PL=0
MOVL C01792 V=800.0 PL=0
MOVL C01793 V=800.0 PL=0
MOVL C01794 V=800.0 PL=0
MOVL C01795 V=800.0 PL=0
MOVL C01796 V=800.0 PL=0
MOVL C01797 V=800.0 PL=0
MOVL C01798 V=800.0 PL=0
MOVL C01799 V=800.0 PL=0
MOVL C01800 V=800.0 PL=0
MOVL C01801 V=800.0 PL=0
MOVL C01802 V=800.0 PL=0
MOVL C01803 V=800.0 PL=0
MOVL C01804 V=800.0 PL=0
MOVL C01805 V=800.0 PL=0
MOVL C01806 V=800.0 PL=0
MOVL C01807 V=800.0 PL=0
MOVL C01808 V=800.0 PL=0
MOVL C01809 V=800.0 PL=0
MOVL C01810 V=800.0 PL=0
MOVL C01811 V=800.0 PL=0
MOVL C01812 V=800.0 PL=0
MOVL C01813 V=800.0 PL=0
MOVL C01814 V=800.0 PL=0
MOVL C01815 V=800.0 PL=0
MOVL C01816 V=800.0 PL=0
MOVL C01817 V=800.0 PL=0
MOVL C01818 V=800.0 PL=0
MOVL C01819 V=800.0 PL=0
MOVL C01820 V=800.0 PL=0
MOVL C01821 V=800.0 PL=0
MOVL C01822 V=800.0 PL=0
MOVL C01823 V=800.0 PL=0
MOVL C01824 V=800.0 PL=0
MOVL C01825 V=800.0 PL=0
MOVL C01826 V=800.0 PL=0
MOVL C01827 V=800.0 PL=0
MOVL C01828 V=800.0 PL=0
MOVL C01829 V=800.0 PL=0
MOVL C01830 V=800.0 PL=0
MOVL C01831 V=800.0 PL=0
MOVL C01832 V=800.0 PL=0
MOVL C01833 V=800.0 PL=0
MOVL C01834 V=800.0 PL=0
MOVL C01835 V=800.0 PL=0
MOVL C01836 V=800.0 PL=0
MOVL C01837 V=800.0 PL=0
MOVL C01838 V=800.0 PL=0
MOVL C01839 V=800.0 PL=0
MOVL C01840 V=800.0 PL=0
MOVL C01841 V=800.0 PL=0
MOVL C01842 V=800.0 PL=0
MOVL C01843 V=800.0 PL=0
MOVL C01844 V=800.0 PL=0
MOVL C01845 V=800.0 PL=0
MOVL C01846 V=800.0 PL=0
MOVL C01847 V=800.0 PL=0
MOVL C01848 V=800.0 PL=0
MOVL C01849 V=800.0 PL=0
MOVL C01850 V=800.0 PL=0
MOVL C01851 V=800.0 PL=0
MOVL C01852 V=800.0 PL=0
MOVL C01853 V=800.0 PL=0
MOVL C01854 V=800.0 PL=0
MOVL C01855 V=800.0 PL=0
MOVL C01856 V=800.0 PL=0
MOVL C01857 V=800.0 PL=0
MOVL C01858 V=800.0 PL=0
MOVL C01859 V=800.0 PL=0
MOVL C01860 V=800.0 PL=0
MOVL C01861 V=800.0 PL=0
MOVL C01862 V=800.0 PL=0
MOVL C01863 V=800.0 PL=0
MOVL C01864 V=800.0 PL=0
MOVL C01865 V=800.0 PL=0
MOVL C01866 V=800.0 PL=0
MOVL C01867 V=800.0 PL=0
MOVL C01868 V=800.0 PL=0
MOVL C01869 V=800.0 PL=0
MOVL C01870 V=800.0 PL=0
MOVL C01871 V=800.0 PL=0
MOVL C01872 V=800.0 PL=0
MOVL C01873 V=800.0 PL=0
MOVL C01874 V=800.0 PL=0
MOVL C01875 V=800.0 PL=0
MOVL C01876 V=800.0 PL=0
MOVL C01877 V=800.0 PL=0
MOVL C01878 V=800.0 PL=0
MOVL C01879 V=800.0 PL=0
MOVL C01880 V=800.0 PL=0
MOVL C01881 V=800.0 PL=0
MOVL C01882 V=800.0 PL=0
MOVL C01883 V=800.0 PL=0
MOVL C01884 V=800.0 PL=0
MOVL C01885 V=800.0 PL=0
MOVL C01886 V=800.0 PL=0
MOVL C01887 V=800.0 PL=0
MOVL C01888 V=800.0 PL=0
MOVL C01889 V=800.0 PL=0
MOVL C01890 V=800.0 PL=0
MOVL C01891 V=800.0 PL=0
MOVL C01892 V=800.0 PL=0
MOVL C01893 V=800.0 PL=0
MOVL C01894 V=800.0 PL=0
MOVL C01895 V=800.0 PL=0
MOVL C01896 V=800.0 PL=0
MOVL C01897 V=800.0 PL=0
MOVL C01898 V=800.0 PL=0
MOVL C01899 V=800.0 PL=0
MOVL C01900 V=800.0 PL=0
MOVL C01901 V=800.0 PL=0
MOVL C01902 V=800.0 PL=0
MOVL C01903 V=800.0 PL=0
MOVL C01904 V=800.0 PL=0
MOVL C01905 V=800.0 PL=0
MOVL C01906 V=800.0 PL=0
MOVL C01907 V=800.0 PL=0
MOVL C01908 V=800.0 PL=0
MOVL C01909 V=800.0 PL=0
MOVL C01910 V=800.0 PL=0
MOVL C01911 V=800.0 PL=0
MOVL C01912 V=800.0 PL=0
MOVL C01913 V=800.0 PL=0
MOVL C01914 V=800.0 PL=0
MOVL C01915 V=800.0 PL=0
MOVL C01916 V=800.0 PL=0
MOVL C01917 V=800.0 PL=0
MOVL C01918 V=800.0 PL=0
MOVL C01919 V=800.0 PL=0
MOVL C01920 V=800.0 PL=0
MOVL C01921 V=800.0 PL=0
MOVL C01922 V=800.0 PL=0
MOVL C01923 V=800.0 PL=0
MOVL C01924 V=800.0 PL=0
MOVL C01925 V=800.0 PL=0
MOVL C01926 V=800.0 PL=0
MOVL C01927 V=800.0 PL=0
MOVL C01928 V=800.0 PL=0
MOVL C01929 V=800.0 PL=0
MOVL C01930 V=800.0 PL=0
MOVL C01931 V=800.0 PL=0
MOVL C01932 V=800.0 PL=0
MOVL C01933 V=800.0 PL=0
MOVL C01934 V=800.0 PL=0
MOVL C01935 V=800.0 PL=0
MOVL C01936 V=800.0 PL=0
MOVL C01937 V=800.0 PL=0
MOVL C01938 V=800.0 PL=0
MOVL C01939 V=800.0 PL=0
MOVL C01940 V=800.0 PL=0
MOVL C01941 V=800.0 PL=0
MOVL C01942 V=800.0 PL=0
MOVL C01943 V=800.0 PL=0
MOVL C01944 V=800.0 PL=0
MOVL C01945 V=800.0 PL=0
MOVL C01946 V=800.0 PL=0
MOVL C01947 V=800.0 PL=0
MOVL C01948 V=800.0 PL=0
MOVL C01949 V=800.0 PL=0
MOVL C01950 V=800.0 PL=0
MOVL C01951 V=800.0 PL=0
MOVL C01952 V=800.0 PL=0
MOVL C01953 V=800.0 PL=0
MOVL C01954 V=800.0 PL=0
MOVL C01955 V=800.0 PL=0
MOVL C01956 V=800.0 PL=0
MOVL C01957 V=800.0 PL=0
MOVL C01958 V=800.0 PL=0
MOVL C01959 V=800.0 PL=0
MOVL C01960 V=800.0 PL=0
MOVL C01961 V=800.0 PL=0
MOVL C01962 V=800.0 PL=0
MOVL C01963 V=800.0 PL=0
MOVL C01964 V=800.0 PL=0
MOVL C01965 V=800.0 PL=0
MOVL C01966 V=800.0 PL=0
MOVL C01967 V=800.0 PL=0
MOVL C01968 V=800.0 PL=0
MOVL C01969 V=800.0 PL=0
MOVL C01970 V=800.0 PL=0
MOVL C01971 V=800.0 PL=0
MOVL C01972 V=800.0 PL=0
MOVL C01973 V=800.0 PL=0
MOVL C01974 V=800.0 PL=0
MOVL C01975 V=800.0 PL=0
MOVL C01976 V=800.0 PL=0
MOVL C01977 V=800.0 PL=0
MOVL C01978 V=800.0 PL=0
MOVL C01979 V=800.0 PL=0
MOVL C01980 V=800.0 PL=0
MOVL C01981 V=800.0 PL=0
MOVL C01982 V=800.0 PL=0
MOVL C01983 V=800.0 PL=0
MOVL C01984 V=800.0 PL=0
MOVL C01985 V=800.0 PL=0
MOVL C01986 V=800.0 PL=0
MOVL C01987 V=800.0 PL=0
MOVL C01988 V=800.0 PL=0
MOVL C01989 V=800.0 PL=0
MOVL C01990 V=800.0 PL=0
MOVL C01991 V=800.0 PL=0
MOVL C01992 V=800.0 PL=0
MOVL C01993 V=800.0 PL=0
MOVL C01994 V=800.0 PL=0
MOVL C01995 V=800.0 PL=0
MOVL C01996 V=800.0 PL=0
MOVL C01997 V=800.0 PL=0
MOVL C01998 V=800.0 PL=0
MOVL C01999 V=800.0 PL=0
MOVL C02000 V=800.0 PL=0
MOVL C02001 V=800.0 PL=0
MOVL C02002 V=800.0 PL=0
MOVL C02003 V=800.0 PL=0
MOVL C02004 V=800.0 PL=0
MOVL C02005 V=800.0 PL=0
MOVL C02006 V=800.0 PL=0
MOVL C02007 V=800.0 PL=0
MOVL C02008 V=800.0 PL=0
MOVL C02009 V=800.0 PL=0
MOVL C02010 V=800.0 PL=0
MOVL C02011 V=800.0 PL=0
MOVL C02012 V=800.0 PL=0
MOVL C02013 V=800.0 PL=0
MOVL C02014 V=800.0 PL=0
MOVL C02015 V=800.0 PL=0
MOVL C02016 V=800.0 PL=0
MOVL C02017 V=800.0 PL=0
MOVL C02018 V=800.0 PL=0
MOVL C02019 V=800.0 PL=0
MOVL C02020 V=800.0 PL=0
MOVL C02021 V=800.0 PL=0
MOVL C02022 V=800.0 PL=0
MOVL C02023 V=800.0 PL=0
MOVL C02024 V=800.0 PL=0
MOVL C02025 V=800.0 PL=0
MOVL C02026 V=800.0 PL=0
MOVL C02027 V=800.0 PL=0
MOVL C02028 V=800.0 PL=0
MOVL C02029 V=800.0 PL=0
MOVL C02030 V=800.0 PL=0
MOVL C02031 V=800.0 PL=0
MOVL C02032 V=800.0 PL=0
MOVL C02033 V=800.0 PL=0
MOVL C02034 V=800.0 PL=0
MOVL C02035 V=800.0 PL=0
MOVL C02036 V=800.0 PL=0
MOVL C02037 V=800.0 PL=0
MOVL C02038 V=800.0 PL=0
MOVL C02039 V=800.0 PL=0
MOVL C02040 V=800.0 PL=0
MOVL C02041 V=800.0 PL=0
MOVL C02042 V=800.0 PL=0
MOVL C02043 V=800.0 PL=0
MOVL C02044 V=800.0 PL=0
MOVL C02045 V=800.0 PL=0
MOVL C02046 V=800.0 PL=0
MOVL C02047 V=800.0 PL=0
MOVL C02048 V=800.0 PL=0
MOVL C02049 V=800.0 PL=0
MOVL C02050 V=800.0 PL=0
MOVL C02051 V=800.0 PL=0
MOVL C02052 V=800.0 PL=0
MOVL C02053 V=800.0 PL=0
MOVL C02054 V=800.0 PL=0
MOVL C02055 V=800.0 PL=0
MOVL C02056 V=800.0 PL=0
MOVL C02057 V=800.0 PL=0
MOVL C02058 V=800.0 PL=0
MOVL C02059 V=800.0 PL=0
MOVL C02060 V=800.0 PL=0
MOVL C02061 V=800.0 PL=0
MOVL C02062 V=800.0 PL=0
MOVL C02063 V=800.0 PL=0
MOVL C02064 V=800.0 PL=0
MOVL C02065 V=800.0 PL=0
MOVL C02066 V=800.0 PL=0
MOVL C02067 V=800.0 PL=0
MOVL C02068 V=800.0 PL=0
MOVL C02069 V=800.0 PL=0
MOVL C02070 V=800.0 PL=0
MOVL C02071 V=800.0 PL=0
MOVL C02072 V=800.0 PL=0
MOVL C02073 V=800.0 PL=0
MOVL C02074 V=800.0 PL=0
MOVL C02075 V=800.0 PL=0
MOVL C02076 V=800.0 PL=0
MOVL C02077 V=800.0 PL=0
MOVL C02078 V=800.0 PL=0
MOVL C02079 V=800.0 PL=0
MOVL C02080 V=800.0 PL=0
MOVL C02081 V=800.0 PL=0
MOVL C02082 V=800.0 PL=0
MOVL C02083 V=800.0 PL=0
MOVL C02084 V=800.0 PL=0
MOVL C02085 V=800.0 PL=0
MOVL C02086 V=800.0 PL=0
MOVL C02087 V=800.0 PL=0
MOVL C02088 V=800.0 PL=0
MOVL C02089 V=800.0 PL=0
MOVL C02090 V=800.0 PL=0
MOVL C02091 V=800.0 PL=0
MOVL C02092 V=800.0 PL=0
MOVL C02093 V=800.0 PL=0
MOVL C02094 V=800.0 PL=0
MOVL C02095 V=800.0 PL=0
MOVL C02096 V=800.0 PL=0
MOVL C02097 V=800.0 PL=0
MOVL C02098 V=800.0 PL=0
MOVL C02099 V=800.0 PL=0
MOVL C02100 V=800.0 PL=0
MOVL C02101 V=800.0 PL=0
MOVL C02102 V=800.0 PL=0
MOVL C02103 V=800.0 PL=0
MOVL C02104 V=800.0 PL=0
MOVL C02105 V=800.0 PL=0
MOVL C02106 V=800.0 PL=0
MOVL C02107 V=800.0 PL=0
